LIN {X 0,Y 236.008,Z 310.681,A -85,B 0,C 180,E1 -19500.944,E2 -19500.944} C_VEL
LIN {X 0,Y 236.836,Z 313.931,A -85,B 0,C 180,E1 -19501.282,E2 -19501.282} C_VEL
LIN {X 0,Y 239.415,Z 324.062,A -85,B 0,C 180,E1 -19502.528,E2 -19502.528} C_VEL
LIN {X 0,Y 241.181,Z 333.604,A -85,B 0,C 180,E1 -19503.852,E2 -19503.852} C_VEL
LIN {X 0,Y 242.176,Z 341.797,A -85,B 0,C 180,E1 -19505.138,E2 -19505.138} C_VEL
LIN {X 0,Y 242.615,Z 349.643,A -85,B 0,C 180,E1 -19506.53,E2 -19506.53} C_VEL
LIN {X 0,Y 242.455,Z 357.246,A -85,B 0,C 180,E1 -19508.066,E2 -19508.066} C_VEL
LIN {X 0,Y 241.956,Z 362.587,A -85,B 0,C 180,E1 -19509.279,E2 -19509.279} C_VEL
LIN {X 0,Y 240.306,Z 368.641,A -85,B 0,C 180,E1 -19510.793,E2 -19510.793} C_VEL
LIN {X 0,Y 238.573,Z 374.082,A -85,B 0,C 180,E1 -19512.428,E2 -19512.428} C_VEL
LIN {X 0,Y 236.726,Z 379.604,A -85,B 0,C 180,E1 -19514.505,E2 -19514.505} C_VEL
LIN {X 0,Y 235.064,Z 384.766,A -85,B 0,C 180,E1 -19517.044,E2 -19517.044} C_VEL
LIN {X 0,Y 233.873,Z 388.583,A -85,B 0,C 180,E1 -19519.615,E2 -19519.615} C_VEL
LIN {X 0,Y 233.308,Z 390.355,A -85,B 0,C 180,E1 -19521.34,E2 -19521.34} C_VEL
LIN {X 0,Y 232.985,Z 391.647,A -85,B 0,C 180,E1 -19523.072,E2 -19523.072} C_VEL
LIN {X 0,Y 232.787,Z 392.537,A -85,B 0,C 180,E1 -19525.087,E2 -19525.087} C_VEL
LIN {X 0,Y 232.804,Z 392.826,A -85,B 0,C 180,E1 -19526.541,E2 -19526.541} C_VEL
LIN {X 0,Y 232.91,Z 392.585,A -85,B 0,C 180,E1 -19528.273,E2 -19528.273} C_VEL
LIN {X 0,Y 232.953,Z 391.86,A -85,B 0,C 180,E1 -19530.002,E2 -19530.002} C_VEL
LIN {X 0,Y 232.952,Z 390.653,A -85,B 0,C 180,E1 -19531.731,E2 -19531.731} C_VEL
LIN {X 0,Y 232.931,Z 388.936,A -85,B 0,C 180,E1 -19533.462,E2 -19533.462} C_VEL
LIN {X 0,Y 232.977,Z 385.143,A -85,B 0,C 180,E1 -19536.063,E2 -19536.063} C_VEL
LIN {X 0,Y 233.32,Z 379.947,A -85,B 0,C 180,E1 -19538.664,E2 -19538.664} C_VEL
LIN {X 0,Y 233.786,Z 374.337,A -85,B 0,C 180,E1 -19540.832,E2 -19540.832} C_VEL
LIN {X 0,Y 234.62,Z 367.267,A -85,B 0,C 180,E1 -19542.985,E2 -19542.985} C_VEL
LIN {X 0,Y 235.626,Z 359.155,A -85,B 0,C 180,E1 -19544.91,E2 -19544.91} C_VEL
LIN {X 0,Y 236.286,Z 352.615,A -85,B 0,C 180,E1 -19546.194,E2 -19546.194} C_VEL
LIN {X 0,Y 236.114,Z 344.809,A -85,B 0,C 180,E1 -19547.498,E2 -19547.498} C_VEL
LIN {X 0,Y 235.752,Z 335.886,A -85,B 0,C 180,E1 -19548.713,E2 -19548.713} C_VEL
LIN {X 0,Y 235.263,Z 327.406,A -85,B 0,C 180,E1 -19549.64,E2 -19549.64} C_VEL
LIN {X 0,Y 234.318,Z 317.752,A -85,B 0,C 180,E1 -19550.466,E2 -19550.466} C_VEL
LIN {X 0,Y 233.579,Z 311.732,A -85,B 0,C 180,E1 -19550.937,E2 -19550.937} C_VEL
LIN {X 0,Y 234.467,Z 305.559,A -85,B 0,C 180,E1 -19555.938,E2 -19555.938} C_VEL
LIN {X 0,Y 235.489,Z 299.992,A -85,B 0,C 180,E1 -19560.49,E2 -19560.49} C_VEL
LIN {X 0,Y 236.19,Z 296.337,A -85,B 0,C 180,E1 -19563.572,E2 -19563.572} C_VEL
LIN {X 0,Y 236.161,Z 294.216,A -85,B 0,C 180,E1 -19565.432,E2 -19565.432} C_VEL
LIN {X 0,Y 235.471,Z 290.233,A -85,B 0,C 180,E1 -19569.1,E2 -19569.1} C_VEL
LIN {X 0,Y 235.075,Z 288.016,A -85,B 0,C 180,E1 -19571.3,E2 -19571.3} C_VEL
LIN {X 0,Y 234.899,Z 288.035,A -85,B 0,C 180,E1 -19576.514,E2 -19576.514} C_VEL
LIN {X 0,Y 234.93,Z 288.031,A -85,B 0,C 180,E1 -19581.078,E2 -19581.078} C_VEL
LIN {X 0,Y 234.942,Z 288.032,A -85,B 0,C 180,E1 -19585.361,E2 -19585.361} C_VEL
LIN {X 0,Y 234.943,Z 288.029,A -85,B 0,C 180,E1 -19589.431,E2 -19589.431} C_VEL
LIN {X 0,Y 235.006,Z 288.023,A -85,B 0,C 180,E1 -19593.792,E2 -19593.792} C_VEL
LIN {X 0,Y 234.98,Z 288.022,A -85,B 0,C 180,E1 -19598.964,E2 -19598.964} C_VEL
LIN {X 0,Y 235.067,Z 288.018,A -85,B 0,C 180,E1 -19603.09,E2 -19603.09} C_VEL
LIN {X 0,Y 235.106,Z 288.003,A -85,B 0,C 180,E1 -19607.919,E2 -19607.919} C_VEL
LIN {X 0,Y 235.328,Z 287.982,A -85,B 0,C 180,E1 -19611.409,E2 -19611.409} C_VEL
LIN {X 0,Y 235.375,Z 287.978,A -85,B 0,C 180,E1 -19613.138,E2 -19613.138} C_VEL
LIN {X 0,Y 235.603,Z 287.945,A -85,B 0,C 180,E1 -19618.288,E2 -19618.288} C_VEL
LIN {X 0,Y 235.603,Z 287.946,A -85,B 0,C 180,E1 -19621.706,E2 -19621.706} C_VEL
LIN {X 0,Y 235.411,Z 287.971,A -85,B 0,C 180,E1 -19626.855,E2 -19626.855} C_VEL
LIN {X 0,Y 235.243,Z 287.989,A -85,B 0,C 180,E1 -19630.323,E2 -19630.323} C_VEL
LIN {X 0,Y 235.116,Z 288.009,A -85,B 0,C 180,E1 -19635.603,E2 -19635.603} C_VEL
LIN {X 0,Y 235.012,Z 288.02,A -85,B 0,C 180,E1 -19639.202,E2 -19639.202} C_VEL
LIN {X 0,Y 234.963,Z 288.023,A -85,B 0,C 180,E1 -19642.879,E2 -19642.879} C_VEL
LIN {X 0,Y 234.97,Z 288.027,A -85,B 0,C 180,E1 -19646.653,E2 -19646.653} C_VEL
LIN {X 0,Y 234.931,Z 288.031,A -85,B 0,C 180,E1 -19650.564,E2 -19650.564} C_VEL
LIN {X 0,Y 234.958,Z 288.027,A -85,B 0,C 180,E1 -19654.629,E2 -19654.629} C_VEL
LIN {X 0,Y 234.994,Z 288.025,A -85,B 0,C 180,E1 -19658.957,E2 -19658.957} C_VEL
LIN {X 0,Y 234.991,Z 288.027,A -85,B 0,C 180,E1 -19663.457,E2 -19663.457} C_VEL
LIN {X 0,Y 234.99,Z 288.024,A -85,B 0,C 180,E1 -19666.535,E2 -19666.535} C_VEL
LIN {X 0,Y 234.948,Z 288.032,A -85,B 0,C 180,E1 -19671.082,E2 -19671.082} C_VEL
LIN {X 0,Y 234.952,Z 288.03,A -85,B 0,C 180,E1 -19675.363,E2 -19675.363} C_VEL
LIN {X 0,Y 234.959,Z 288.029,A -85,B 0,C 180,E1 -19680.154,E2 -19680.154} C_VEL
LIN {X 0,Y 234.983,Z 288.025,A -85,B 0,C 180,E1 -19683.79,E2 -19683.79} C_VEL
LIN {X 0,Y 234.963,Z 288.028,A -85,B 0,C 180,E1 -19687.998,E2 -19687.998} C_VEL
LIN {X 0,Y 234.735,Z 288.058,A -85,B 0,C 180,E1 -19692.576,E2 -19692.576} C_VEL
LIN {X 0,Y 234.34,Z 288.106,A -85,B 0,C 180,E1 -19696.116,E2 -19696.116} C_VEL
LIN {X 0,Y 234.116,Z 288.347,A -85,B 0,C 180,E1 -19698.307,E2 -19698.307} C_VEL
LIN {X 0,Y 234.103,Z 291.422,A -85,B 0,C 180,E1 -19702.145,E2 -19702.145} C_VEL
LIN {X 0,Y 234.001,Z 292.577,A -85,B 0,C 180,E1 -19703.314,E2 -19703.314} C_VEL
LIN {X 0,Y 236.168,Z 303.411,A -85,B 0,C 180,E1 -19704.234,E2 -19704.234} C_VEL
LIN {X 0,Y 237.327,Z 311.672,A -85,B 0,C 180,E1 -19705.114,E2 -19705.114} C_VEL
LIN {X 0,Y 238.306,Z 321.335,A -85,B 0,C 180,E1 -19706.405,E2 -19706.405} C_VEL
LIN {X 0,Y 237.452,Z 329.525,A -85,B 0,C 180,E1 -19707.665,E2 -19707.665} C_VEL
LIN {X 0,Y 236.487,Z 337.321,A -85,B 0,C 180,E1 -19709.146,E2 -19709.146} C_VEL
LIN {X 0,Y 235.36,Z 346.28,A -85,B 0,C 180,E1 -19711.281,E2 -19711.281} C_VEL
LIN {X 0,Y 234.486,Z 353.183,A -85,B 0,C 180,E1 -19713.434,E2 -19713.434} C_VEL
LIN {X 0,Y 233.98,Z 357.734,A -85,B 0,C 180,E1 -19715.168,E2 -19715.168} C_VEL
LIN {X 0,Y 233.523,Z 361.536,A -85,B 0,C 180,E1 -19716.912,E2 -19716.912} C_VEL
LIN {X 0,Y 232.998,Z 365.862,A -85,B 0,C 180,E1 -19719.547,E2 -19719.547} C_VEL
LIN {X 0,Y 232.736,Z 368.898,A -85,B 0,C 180,E1 -19722.201,E2 -19722.201} C_VEL
LIN {X 0,Y 232.797,Z 370.803,A -85,B 0,C 180,E1 -19724.987,E2 -19724.987} C_VEL
LIN {X 0,Y 233.038,Z 371.385,A -85,B 0,C 180,E1 -19727.55,E2 -19727.55} C_VEL
LIN {X 0,Y 233.453,Z 371.103,A -85,B 0,C 180,E1 -19729.336,E2 -19729.336} C_VEL
LIN {X 0,Y 234.146,Z 370.082,A -85,B 0,C 180,E1 -19731.502,E2 -19731.502} C_VEL
LIN {X 0,Y 235.525,Z 367.076,A -85,B 0,C 180,E1 -19734.69,E2 -19734.69} C_VEL
LIN {X 0,Y 237.062,Z 363.279,A -85,B 0,C 180,E1 -19737.213,E2 -19737.213} C_VEL
LIN {X 0,Y 238.439,Z 359.51,A -85,B 0,C 180,E1 -19739.097,E2 -19739.097} C_VEL
LIN {X 0,Y 239.916,Z 355.184,A -85,B 0,C 180,E1 -19740.837,E2 -19740.837} C_VEL
LIN {X 0,Y 241.768,Z 349.341,A -85,B 0,C 180,E1 -19742.728,E2 -19742.728} C_VEL
LIN {X 0,Y 243.49,Z 343.538,A -85,B 0,C 180,E1 -19744.249,E2 -19744.249} C_VEL
LIN {X 0,Y 245.449,Z 336.245,A -85,B 0,C 180,E1 -19745.811,E2 -19745.811} C_VEL
LIN {X 0,Y 245.573,Z 333.35,A -85,B 0,C 180,E1 -19746.445,E2 -19746.445} C_VEL
LIN {X 0,Y 244.381,Z 324.378,A -85,B 0,C 180,E1 -19748.274,E2 -19748.274} C_VEL
LIN {X 0,Y 242.509,Z 315.823,A -85,B 0,C 180,E1 -19749.832,E2 -19749.832} C_VEL
LIN {X 0,Y 240.136,Z 307.625,A -85,B 0,C 180,E1 -19751.189,E2 -19751.189} C_VEL
LIN {X 0,Y 236.731,Z 298.443,A -85,B 0,C 180,E1 -19752.592,E2 -19752.592} C_VEL
LIN {X 0,Y 235.009,Z 293.938,A -85,B 0,C 180,E1 -19753.227,E2 -19753.227} C_VEL
LIN {X 0,Y 234.961,Z 293.585,A -85,B 0,C 180,E1 -19753.299,E2 -19753.299} C_VEL
LIN {X 0,Y 235.134,Z 291.455,A -85,B 0,C 180,E1 -19756.576,E2 -19756.576} C_VEL
LIN {X 0,Y 235.094,Z 290.036,A -85,B 0,C 180,E1 -19758.882,E2 -19758.882} C_VEL
LIN {X 0,Y 235.006,Z 288.731,A -85,B 0,C 180,E1 -19761.101,E2 -19761.101} C_VEL
LIN {X 0,Y 234.937,Z 288.037,A -85,B 0,C 180,E1 -19763.866,E2 -19763.866} C_VEL
LIN {X 0,Y 234.943,Z 288.032,A -85,B 0,C 180,E1 -19767.427,E2 -19767.427} C_VEL
LIN {X 0,Y 234.919,Z 288.033,A -85,B 0,C 180,E1 -19771.406,E2 -19771.406} C_VEL
LIN {X 0,Y 234.963,Z 288.03,A -85,B 0,C 180,E1 -19775.248,E2 -19775.248} C_VEL
LIN {X 0,Y 234.983,Z 288.023,A -85,B 0,C 180,E1 -19778.971,E2 -19778.971} C_VEL
LIN {X 0,Y 235.082,Z 288.011,A -85,B 0,C 180,E1 -19783.062,E2 -19783.062} C_VEL
LIN {X 0,Y 235.13,Z 288.01,A -85,B 0,C 180,E1 -19787.926,E2 -19787.926} C_VEL
LIN {X 0,Y 235.309,Z 287.988,A -85,B 0,C 180,E1 -19791.415,E2 -19791.415} C_VEL
LIN {X 0,Y 235.347,Z 287.975,A -85,B 0,C 180,E1 -19793.143,E2 -19793.143} C_VEL
LIN {X 0,Y 235.586,Z 287.945,A -85,B 0,C 180,E1 -19798.294,E2 -19798.294} C_VEL
LIN {X 0,Y 235.586,Z 287.945,A -85,B 0,C 180,E1 -19801.713,E2 -19801.713} C_VEL
LIN {X 0,Y 235.397,Z 287.97,A -85,B 0,C 180,E1 -19806.862,E2 -19806.862} C_VEL
LIN {X 0,Y 235.246,Z 287.996,A -85,B 0,C 180,E1 -19810.329,E2 -19810.329} C_VEL
LIN {X 0,Y 235.107,Z 288.012,A -85,B 0,C 180,E1 -19815.61,E2 -19815.61} C_VEL
LIN {X 0,Y 235.002,Z 288.025,A -85,B 0,C 180,E1 -19819.209,E2 -19819.209} C_VEL
LIN {X 0,Y 234.941,Z 288.036,A -85,B 0,C 180,E1 -19822.888,E2 -19822.888} C_VEL
LIN {X 0,Y 234.94,Z 288.037,A -85,B 0,C 180,E1 -19826.664,E2 -19826.664} C_VEL
LIN {X 0,Y 234.895,Z 288.046,A -85,B 0,C 180,E1 -19830.576,E2 -19830.576} C_VEL
LIN {X 0,Y 234.957,Z 288.038,A -85,B 0,C 180,E1 -19834.636,E2 -19834.636} C_VEL
LIN {X 0,Y 234.993,Z 288.035,A -85,B 0,C 180,E1 -19836.153,E2 -19836.153} C_VEL
LIN {X 0,Y 235.324,Z 290.078,A -85,B 0,C 180,E1 -19839.063,E2 -19839.063} C_VEL
LIN {X 0,Y 235.81,Z 293.316,A -85,B 0,C 180,E1 -19843.277,E2 -19843.277} C_VEL
LIN {X 0,Y 236.483,Z 297.318,A -85,B 0,C 180,E1 -19847.988,E2 -19847.988} C_VEL
LIN {X 0,Y 237.095,Z 300.545,A -85,B 0,C 180,E1 -19851.505,E2 -19851.505} C_VEL
LIN {X 0,Y 237.449,Z 303.212,A -85,B 0,C 180,E1 -19854.2,E2 -19854.2} C_VEL
LIN {X 0,Y 236.801,Z 304.253,A -85,B 0,C 180,E1 -19855.103,E2 -19855.103} C_VEL
LIN {X 0,Y 233.819,Z 306.165,A -85,B 0,C 180,E1 -19856.484,E2 -19856.484} C_VEL
LIN {X 0,Y 230.582,Z 308.119,A -85,B 0,C 180,E1 -19857.893,E2 -19857.893} C_VEL
LIN {X 0,Y 229.602,Z 309.245,A -85,B 0,C 180,E1 -19858.83,E2 -19858.83} C_VEL
LIN {X 0,Y 229.293,Z 310.304,A -85,B 0,C 180,E1 -19859.784,E2 -19859.784} C_VEL
LIN {X 0,Y 230.185,Z 313.716,A -85,B 0,C 180,E1 -19860.165,E2 -19860.165} C_VEL
LIN {X 0,Y 232.856,Z 324.19,A -85,B 0,C 180,E1 -19861.531,E2 -19861.531} C_VEL
LIN {X 0,Y 234.553,Z 333.427,A -85,B 0,C 180,E1 -19862.882,E2 -19862.882} C_VEL
LIN {X 0,Y 235.447,Z 340.923,A -85,B 0,C 180,E1 -19864.102,E2 -19864.102} C_VEL
LIN {X 0,Y 236.011,Z 349.022,A -85,B 0,C 180,E1 -19865.598,E2 -19865.598} C_VEL
LIN {X 0,Y 235.901,Z 356.764,A -85,B 0,C 180,E1 -19867.216,E2 -19867.216} C_VEL
LIN {X 0,Y 235.274,Z 362.992,A -85,B 0,C 180,E1 -19868.693,E2 -19868.693} C_VEL
LIN {X 0,Y 233.628,Z 368.826,A -85,B 0,C 180,E1 -19870.222,E2 -19870.222} C_VEL
LIN {X 0,Y 231.835,Z 374.177,A -85,B 0,C 180,E1 -19871.9,E2 -19871.9} C_VEL
LIN {X 0,Y 229.886,Z 379.621,A -85,B 0,C 180,E1 -19874.032,E2 -19874.032} C_VEL
LIN {X 0,Y 228.141,Z 384.711,A -85,B 0,C 180,E1 -19876.644,E2 -19876.644} C_VEL
LIN {X 0,Y 226.878,Z 388.454,A -85,B 0,C 180,E1 -19879.291,E2 -19879.291} C_VEL
LIN {X 0,Y 226.285,Z 390.169,A -85,B 0,C 180,E1 -19881.069,E2 -19881.069} C_VEL
LIN {X 0,Y 225.927,Z 391.401,A -85,B 0,C 180,E1 -19882.855,E2 -19882.855} C_VEL
LIN {X 0,Y 225.706,Z 392.282,A -85,B 0,C 180,E1 -19885.167,E2 -19885.167} C_VEL
LIN {X 0,Y 225.709,Z 392.49,A -85,B 0,C 180,E1 -19886.432,E2 -19886.432} C_VEL
LIN {X 0,Y 225.838,Z 392.227,A -85,B 0,C 180,E1 -19888.219,E2 -19888.219} C_VEL
LIN {X 0,Y 225.882,Z 391.447,A -85,B 0,C 180,E1 -19890.002,E2 -19890.002} C_VEL
LIN {X 0,Y 225.882,Z 390.182,A -85,B 0,C 180,E1 -19891.785,E2 -19891.785} C_VEL
LIN {X 0,Y 225.789,Z 387.389,A -85,B 0,C 180,E1 -19894.352,E2 -19894.352} C_VEL
LIN {X 0,Y 225.918,Z 384.546,A -85,B 0,C 180,E1 -19896.253,E2 -19896.253} C_VEL
LIN {X 0,Y 226.11,Z 381.21,A -85,B 0,C 180,E1 -19898.043,E2 -19898.043} C_VEL
LIN {X 0,Y 226.472,Z 377.155,A -85,B 0,C 180,E1 -19899.83,E2 -19899.83} C_VEL
LIN {X 0,Y 227.131,Z 370.824,A -85,B 0,C 180,E1 -19902.058,E2 -19902.058} C_VEL
LIN {X 0,Y 227.879,Z 364.62,A -85,B 0,C 180,E1 -19903.831,E2 -19903.831} C_VEL
LIN {X 0,Y 228.776,Z 358.107,A -85,B 0,C 180,E1 -19905.367,E2 -19905.367} C_VEL
LIN {X 0,Y 229.258,Z 352.645,A -85,B 0,C 180,E1 -19906.475,E2 -19906.475} C_VEL
LIN {X 0,Y 229.055,Z 343.894,A -85,B 0,C 180,E1 -19907.974,E2 -19907.974} C_VEL
LIN {X 0,Y 228.8,Z 336.258,A -85,B 0,C 180,E1 -19909.05,E2 -19909.05} C_VEL
LIN {X 0,Y 228.248,Z 326.901,A -85,B 0,C 180,E1 -19910.111,E2 -19910.111} C_VEL
LIN {X 0,Y 227.293,Z 317.696,A -85,B 0,C 180,E1 -19910.93,E2 -19910.93} C_VEL
LIN {X 0,Y 226.538,Z 311.466,A -85,B 0,C 180,E1 -19911.381,E2 -19911.381} C_VEL
LIN {X 0,Y 227.302,Z 306.394,A -85,B 0,C 180,E1 -19915.652,E2 -19915.652} C_VEL
LIN {X 0,Y 228.394,Z 300.678,A -85,B 0,C 180,E1 -19920.499,E2 -19920.499} C_VEL
LIN {X 0,Y 229.108,Z 297.178,A -85,B 0,C 180,E1 -19923.518,E2 -19923.518} C_VEL
LIN {X 0,Y 229.089,Z 294.828,A -85,B 0,C 180,E1 -19925.656,E2 -19925.656} C_VEL
LIN {X 0,Y 228.228,Z 289.995,A -85,B 0,C 180,E1 -19930.293,E2 -19930.293} C_VEL
LIN {X 0,Y 227.996,Z 288.898,A -85,B 0,C 180,E1 -19931.512,E2 -19931.512} C_VEL
LIN {X 0,Y 227.846,Z 288.914,A -85,B 0,C 180,E1 -19935.192,E2 -19935.192} C_VEL
LIN {X 0,Y 227.838,Z 288.918,A -85,B 0,C 180,E1 -19939.623,E2 -19939.623} C_VEL
LIN {X 0,Y 227.893,Z 288.909,A -85,B 0,C 180,E1 -19944.127,E2 -19944.127} C_VEL
LIN {X 0,Y 227.882,Z 288.906,A -85,B 0,C 180,E1 -19948.377,E2 -19948.377} C_VEL
LIN {X 0,Y 227.898,Z 288.907,A -85,B 0,C 180,E1 -19952.444,E2 -19952.444} C_VEL
LIN {X 0,Y 227.917,Z 288.902,A -85,B 0,C 180,E1 -19956.365,E2 -19956.365} C_VEL
LIN {X 0,Y 227.925,Z 288.902,A -85,B 0,C 180,E1 -19960.17,E2 -19960.17} C_VEL
LIN {X 0,Y 228.031,Z 288.891,A -85,B 0,C 180,E1 -19963.893,E2 -19963.893} C_VEL
LIN {X 0,Y 228.064,Z 288.881,A -85,B 0,C 180,E1 -19967.54,E2 -19967.54} C_VEL
LIN {X 0,Y 228.26,Z 288.864,A -85,B 0,C 180,E1 -19971.141,E2 -19971.141} C_VEL
LIN {X 0,Y 228.325,Z 288.858,A -85,B 0,C 180,E1 -19972.925,E2 -19972.925} C_VEL
LIN {X 0,Y 228.561,Z 288.822,A -85,B 0,C 180,E1 -19978.235,E2 -19978.235} C_VEL
LIN {X 0,Y 228.562,Z 288.823,A -85,B 0,C 180,E1 -19981.759,E2 -19981.759} C_VEL
LIN {X 0,Y 228.361,Z 288.849,A -85,B 0,C 180,E1 -19987.068,E2 -19987.068} C_VEL
LIN {X 0,Y 228.169,Z 288.87,A -85,B 0,C 180,E1 -19990.647,E2 -19990.647} C_VEL
LIN {X 0,Y 228.067,Z 288.889,A -85,B 0,C 180,E1 -19994.268,E2 -19994.268} C_VEL
LIN {X 0,Y 228.007,Z 288.897,A -85,B 0,C 180,E1 -19997.949,E2 -19997.949} C_VEL
LIN {X 0,Y 227.932,Z 288.9,A -85,B 0,C 180,E1 -20002.325,E2 -20002.325} C_VEL
LIN {X 0,Y 227.943,Z 288.902,A -85,B 0,C 180,E1 -20006.598,E2 -20006.598} C_VEL
LIN {X 0,Y 227.907,Z 288.906,A -85,B 0,C 180,E1 -20010.291,E2 -20010.291} C_VEL
LIN {X 0,Y 227.888,Z 288.911,A -85,B 0,C 180,E1 -20013.714,E2 -20013.714} C_VEL
LIN {X 0,Y 227.888,Z 288.91,A -85,B 0,C 180,E1 -20018.077,E2 -20018.077} C_VEL
LIN {X 0,Y 227.931,Z 288.904,A -85,B 0,C 180,E1 -20022.709,E2 -20022.709} C_VEL
LIN {X 0,Y 227.923,Z 288.908,A -85,B 0,C 180,E1 -20027.281,E2 -20027.281} C_VEL
LIN {X 0,Y 227.864,Z 288.912,A -85,B 0,C 180,E1 -20031.91,E2 -20031.91} C_VEL
LIN {X 0,Y 227.881,Z 288.911,A -85,B 0,C 180,E1 -20036.369,E2 -20036.369} C_VEL
LIN {X 0,Y 227.909,Z 288.908,A -85,B 0,C 180,E1 -20040.434,E2 -20040.434} C_VEL
LIN {X 0,Y 227.917,Z 288.908,A -85,B 0,C 180,E1 -20044.422,E2 -20044.422} C_VEL
LIN {X 0,Y 227.921,Z 288.907,A -85,B 0,C 180,E1 -20048.281,E2 -20048.281} C_VEL
LIN {X 0,Y 227.668,Z 288.937,A -85,B 0,C 180,E1 -20053.113,E2 -20053.113} C_VEL
LIN {X 0,Y 227.073,Z 289.046,A -85,B 0,C 180,E1 -20058.166,E2 -20058.166} C_VEL
LIN {X 0,Y 226.974,Z 292.656,A -85,B 0,C 180,E1 -20062.791,E2 -20062.791} C_VEL
LIN {X 0,Y 229.271,Z 304.335,A -85,B 0,C 180,E1 -20063.839,E2 -20063.839} C_VEL
LIN {X 0,Y 230.419,Z 312.457,A -85,B 0,C 180,E1 -20064.748,E2 -20064.748} C_VEL
LIN {X 0,Y 231.205,Z 320.636,A -85,B 0,C 180,E1 -20065.858,E2 -20065.858} C_VEL
LIN {X 0,Y 231.077,Z 325.043,A -85,B 0,C 180,E1 -20066.51,E2 -20066.51} C_VEL
LIN {X 0,Y 229.823,Z 334.841,A -85,B 0,C 180,E1 -20068.245,E2 -20068.245} C_VEL
LIN {X 0,Y 228.881,Z 342.581,A -85,B 0,C 180,E1 -20069.998,E2 -20069.998} C_VEL
LIN {X 0,Y 228.019,Z 348.96,A -85,B 0,C 180,E1 -20071.764,E2 -20071.764} C_VEL
LIN {X 0,Y 227.352,Z 354.255,A -85,B 0,C 180,E1 -20073.542,E2 -20073.542} C_VEL
LIN {X 0,Y 226.845,Z 358.671,A -85,B 0,C 180,E1 -20075.331,E2 -20075.331} C_VEL
LIN {X 0,Y 226.377,Z 362.354,A -85,B 0,C 180,E1 -20077.131,E2 -20077.131} C_VEL
LIN {X 0,Y 226.018,Z 365.378,A -85,B 0,C 180,E1 -20078.942,E2 -20078.942} C_VEL
LIN {X 0,Y 225.749,Z 367.747,A -85,B 0,C 180,E1 -20080.763,E2 -20080.763} C_VEL
LIN {X 0,Y 225.632,Z 369.493,A -85,B 0,C 180,E1 -20082.591,E2 -20082.591} C_VEL
LIN {X 0,Y 225.729,Z 371.137,A -85,B 0,C 180,E1 -20085.182,E2 -20085.182} C_VEL
LIN {X 0,Y 226.064,Z 371.688,A -85,B 0,C 180,E1 -20088.11,E2 -20088.11} C_VEL
LIN {X 0,Y 226.529,Z 371.38,A -85,B 0,C 180,E1 -20089.952,E2 -20089.952} C_VEL
LIN {X 0,Y 227.194,Z 370.422,A -85,B 0,C 180,E1 -20091.884,E2 -20091.884} C_VEL
LIN {X 0,Y 227.911,Z 369.033,A -85,B 0,C 180,E1 -20093.63,E2 -20093.63} C_VEL
LIN {X 0,Y 229.383,Z 365.869,A -85,B 0,C 180,E1 -20096.373,E2 -20096.373} C_VEL
LIN {X 0,Y 231.271,Z 361.194,A -85,B 0,C 180,E1 -20099.089,E2 -20099.089} C_VEL
LIN {X 0,Y 233.181,Z 355.971,A -85,B 0,C 180,E1 -20101.323,E2 -20101.323} C_VEL
LIN {X 0,Y 234.93,Z 350.723,A -85,B 0,C 180,E1 -20103.117,E2 -20103.117} C_VEL
LIN {X 0,Y 236.883,Z 344.532,A -85,B 0,C 180,E1 -20104.825,E2 -20104.825} C_VEL
LIN {X 0,Y 238.87,Z 337.589,A -85,B 0,C 180,E1 -20106.379,E2 -20106.379} C_VEL
LIN {X 0,Y 239.035,Z 335.431,A -85,B 0,C 180,E1 -20106.869,E2 -20106.869} C_VEL
LIN {X 0,Y 237.849,Z 325.521,A -85,B 0,C 180,E1 -20109.034,E2 -20109.034} C_VEL
LIN {X 0,Y 236.096,Z 317.291,A -85,B 0,C 180,E1 -20110.625,E2 -20110.625} C_VEL
LIN {X 0,Y 233.545,Z 308.548,A -85,B 0,C 180,E1 -20112.165,E2 -20112.165} C_VEL
LIN {X 0,Y 230.284,Z 299.911,A -85,B 0,C 180,E1 -20113.588,E2 -20113.588} C_VEL
LIN {X 0,Y 228.115,Z 294.568,A -85,B 0,C 180,E1 -20114.413,E2 -20114.413} C_VEL
LIN {X 0,Y 228.023,Z 293.993,A -85,B 0,C 180,E1 -20114.508,E2 -20114.508} C_VEL
LIN {X 0,Y 228.108,Z 292.023,A -85,B 0,C 180,E1 -20117.68,E2 -20117.68} C_VEL
LIN {X 0,Y 227.928,Z 289.589,A -85,B 0,C 180,E1 -20121.931,E2 -20121.931} C_VEL
LIN {X 0,Y 227.886,Z 288.915,A -85,B 0,C 180,E1 -20123.302,E2 -20123.302} C_VEL
LIN {X 0,Y 227.873,Z 288.914,A -85,B 0,C 180,E1 -20126.375,E2 -20126.375} C_VEL
LIN {X 0,Y 227.888,Z 288.912,A -85,B 0,C 180,E1 -20130.438,E2 -20130.438} C_VEL
LIN {X 0,Y 227.909,Z 288.909,A -85,B 0,C 180,E1 -20134.428,E2 -20134.428} C_VEL
LIN {X 0,Y 227.933,Z 288.904,A -85,B 0,C 180,E1 -20138.288,E2 -20138.288} C_VEL
LIN {X 0,Y 228.021,Z 288.889,A -85,B 0,C 180,E1 -20142.828,E2 -20142.828} C_VEL
LIN {X 0,Y 228.079,Z 288.888,A -85,B 0,C 180,E1 -20147.547,E2 -20147.547} C_VEL
LIN {X 0,Y 228.247,Z 288.865,A -85,B 0,C 180,E1 -20151.147,E2 -20151.147} C_VEL
LIN {X 0,Y 228.299,Z 288.854,A -85,B 0,C 180,E1 -20152.93,E2 -20152.93} C_VEL
LIN {X 0,Y 228.544,Z 288.822,A -85,B 0,C 180,E1 -20158.241,E2 -20158.241} C_VEL
LIN {X 0,Y 228.545,Z 288.822,A -85,B 0,C 180,E1 -20161.765,E2 -20161.765} C_VEL
LIN {X 0,Y 228.349,Z 288.849,A -85,B 0,C 180,E1 -20167.075,E2 -20167.075} C_VEL
LIN {X 0,Y 228.164,Z 288.877,A -85,B 0,C 180,E1 -20170.653,E2 -20170.653} C_VEL
LIN {X 0,Y 228.051,Z 288.892,A -85,B 0,C 180,E1 -20176.106,E2 -20176.106} C_VEL
LIN {X 0,Y 227.931,Z 288.906,A -85,B 0,C 180,E1 -20179.829,E2 -20179.829} C_VEL
LIN {X 0,Y 227.89,Z 288.912,A -85,B 0,C 180,E1 -20183.638,E2 -20183.638} C_VEL
LIN {X 0,Y 227.85,Z 288.922,A -85,B 0,C 180,E1 -20187.563,E2 -20187.563} C_VEL
LIN {X 0,Y 227.854,Z 288.922,A -85,B 0,C 180,E1 -20191.628,E2 -20191.628} C_VEL
LIN {X 0,Y 227.979,Z 289.073,A -85,B 0,C 180,E1 -20195.314,E2 -20195.314} C_VEL
LIN {X 0,Y 228.451,Z 292.089,A -85,B 0,C 180,E1 -20199.732,E2 -20199.732} C_VEL
LIN {X 0,Y 228.754,Z 294.17,A -85,B 0,C 180,E1 -20202.528,E2 -20202.528} C_VEL
LIN {X 0,Y 229.419,Z 298.061,A -85,B 0,C 180,E1 -20207.329,E2 -20207.329} C_VEL
LIN {X 0,Y 230.072,Z 301.512,A -85,B 0,C 180,E1 -20211.232,E2 -20211.232} C_VEL
LIN {X 0,Y 230.496,Z 304.747,A -85,B 0,C 180,E1 -20214.6,E2 -20214.6} C_VEL
LIN {X 0,Y 229.965,Z 307.974,A -85,B 0,C 180,E1 -20217.671,E2 -20217.671} C_VEL
LIN {X 0,Y 229.602,Z 309.245,A -85,B 0,C 180,E1 -20218.83,E2 -20218.83} C_VEL
LIN {X 0,Y 229.759,Z 310.473,A -85,B 0,C 180,E1 -20219.478,E2 -20219.478} C_VEL
LIN {X 0,Y 230.705,Z 313.064,A -85,B 0,C 180,E1 -20220.17,E2 -20220.17} C_VEL
LIN {X 0,Y 232.123,Z 317.253,A -85,B 0,C 180,E1 -20220.774,E2 -20220.774} C_VEL
LIN {X 0,Y 232.473,Z 321.036,A -85,B 0,C 180,E1 -20221.139,E2 -20221.139} C_VEL
LIN {X 0,Y 231.641,Z 325.307,A -85,B 0,C 180,E1 -20221.418,E2 -20221.418} C_VEL
LIN {X 0,Y 228.832,Z 333.716,A -85,B 0,C 180,E1 -20222.039,E2 -20222.039} C_VEL
LIN {X 0,Y 228.581,Z 337.299,A -85,B 0,C 180,E1 -20222.511,E2 -20222.511} C_VEL
LIN {X 0,Y 229.384,Z 347.335,A -85,B 0,C 180,E1 -20224.378,E2 -20224.378} C_VEL
LIN {X 0,Y 229.364,Z 355.19,A -85,B 0,C 180,E1 -20226.049,E2 -20226.049} C_VEL
LIN {X 0,Y 228.754,Z 362.606,A -85,B 0,C 180,E1 -20227.864,E2 -20227.864} C_VEL
LIN {X 0,Y 227.495,Z 367.593,A -85,B 0,C 180,E1 -20229.193,E2 -20229.193} C_VEL
LIN {X 0,Y 225.113,Z 374.273,A -85,B 0,C 180,E1 -20231.34,E2 -20231.34} C_VEL
LIN {X 0,Y 223.058,Z 379.638,A -85,B 0,C 180,E1 -20233.529,E2 -20233.529} C_VEL
LIN {X 0,Y 221.774,Z 383.127,A -85,B 0,C 180,E1 -20235.317,E2 -20235.317} C_VEL
LIN {X 0,Y 220.256,Z 387.171,A -85,B 0,C 180,E1 -20238.032,E2 -20238.032} C_VEL
LIN {X 0,Y 219.253,Z 389.985,A -85,B 0,C 180,E1 -20240.78,E2 -20240.78} C_VEL
LIN {X 0,Y 218.864,Z 391.157,A -85,B 0,C 180,E1 -20242.623,E2 -20242.623} C_VEL
LIN {X 0,Y 218.61,Z 392.038,A -85,B 0,C 180,E1 -20245.305,E2 -20245.305} C_VEL
LIN {X 0,Y 218.743,Z 391.866,A -85,B 0,C 180,E1 -20248.161,E2 -20248.161} C_VEL
LIN {X 0,Y 218.814,Z 391.03,A -85,B 0,C 180,E1 -20250.002,E2 -20250.002} C_VEL
LIN {X 0,Y 218.814,Z 389.706,A -85,B 0,C 180,E1 -20251.843,E2 -20251.843} C_VEL
LIN {X 0,Y 218.743,Z 387.861,A -85,B 0,C 180,E1 -20253.687,E2 -20253.687} C_VEL
LIN {X 0,Y 218.747,Z 385.462,A -85,B 0,C 180,E1 -20255.533,E2 -20255.533} C_VEL
LIN {X 0,Y 218.944,Z 382.399,A -85,B 0,C 180,E1 -20257.379,E2 -20257.379} C_VEL
LIN {X 0,Y 219.434,Z 376.391,A -85,B 0,C 180,E1 -20260.148,E2 -20260.148} C_VEL
LIN {X 0,Y 219.994,Z 371.404,A -85,B 0,C 180,E1 -20261.987,E2 -20261.987} C_VEL
LIN {X 0,Y 220.719,Z 365.379,A -85,B 0,C 180,E1 -20263.819,E2 -20263.819} C_VEL
LIN {X 0,Y 221.765,Z 358.054,A -85,B 0,C 180,E1 -20265.629,E2 -20265.629} C_VEL
LIN {X 0,Y 222.237,Z 352.764,A -85,B 0,C 180,E1 -20266.752,E2 -20266.752} C_VEL
LIN {X 0,Y 222.049,Z 343.105,A -85,B 0,C 180,E1 -20268.454,E2 -20268.454} C_VEL
LIN {X 0,Y 221.749,Z 334.464,A -85,B 0,C 180,E1 -20269.681,E2 -20269.681} C_VEL
LIN {X 0,Y 221.197,Z 326.273,A -85,B 0,C 180,E1 -20270.626,E2 -20270.626} C_VEL
LIN {X 0,Y 220.314,Z 317.035,A -85,B 0,C 180,E1 -20271.465,E2 -20271.465} C_VEL
LIN {X 0,Y 219.524,Z 311.153,A -85,B 0,C 180,E1 -20271.917,E2 -20271.917} C_VEL
LIN {X 0,Y 220.441,Z 305.581,A -85,B 0,C 180,E1 -20276.783,E2 -20276.783} C_VEL
LIN {X 0,Y 221.456,Z 300.736,A -85,B 0,C 180,E1 -20281.03,E2 -20281.03} C_VEL
LIN {X 0,Y 222.059,Z 297.866,A -85,B 0,C 180,E1 -20283.591,E2 -20283.591} C_VEL
LIN {X 0,Y 222.02,Z 295.475,A -85,B 0,C 180,E1 -20285.849,E2 -20285.849} C_VEL
LIN {X 0,Y 221.217,Z 290.975,A -85,B 0,C 180,E1 -20290.314,E2 -20290.314} C_VEL
LIN {X 0,Y 220.935,Z 289.778,A -85,B 0,C 180,E1 -20291.701,E2 -20291.701} C_VEL
LIN {X 0,Y 220.786,Z 289.794,A -85,B 0,C 180,E1 -20295.546,E2 -20295.546} C_VEL
LIN {X 0,Y 220.819,Z 289.789,A -85,B 0,C 180,E1 -20300.462,E2 -20300.462} C_VEL
LIN {X 0,Y 220.813,Z 289.791,A -85,B 0,C 180,E1 -20305.044,E2 -20305.044} C_VEL
LIN {X 0,Y 220.881,Z 289.78,A -85,B 0,C 180,E1 -20309.394,E2 -20309.394} C_VEL
LIN {X 0,Y 220.907,Z 289.781,A -85,B 0,C 180,E1 -20313.548,E2 -20313.548} C_VEL
LIN {X 0,Y 220.875,Z 289.778,A -85,B 0,C 180,E1 -20317.55,E2 -20317.55} C_VEL
LIN {X 0,Y 220.939,Z 289.775,A -85,B 0,C 180,E1 -20322.616,E2 -20322.616} C_VEL
LIN {X 0,Y 221.002,Z 289.762,A -85,B 0,C 180,E1 -20327.135,E2 -20327.135} C_VEL
LIN {X 0,Y 221.197,Z 289.743,A -85,B 0,C 180,E1 -20330.856,E2 -20330.856} C_VEL
LIN {X 0,Y 221.26,Z 289.737,A -85,B 0,C 180,E1 -20332.697,E2 -20332.697} C_VEL
LIN {X 0,Y 221.519,Z 289.699,A -85,B 0,C 180,E1 -20338.179,E2 -20338.179} C_VEL
LIN {X 0,Y 221.52,Z 289.7,A -85,B 0,C 180,E1 -20341.815,E2 -20341.815} C_VEL
LIN {X 0,Y 221.296,Z 289.728,A -85,B 0,C 180,E1 -20347.295,E2 -20347.295} C_VEL
LIN {X 0,Y 221.117,Z 289.747,A -85,B 0,C 180,E1 -20350.99,E2 -20350.99} C_VEL
LIN {X 0,Y 221.02,Z 289.765,A -85,B 0,C 180,E1 -20356.626,E2 -20356.626} C_VEL
LIN {X 0,Y 220.895,Z 289.775,A -85,B 0,C 180,E1 -20360.482,E2 -20360.482} C_VEL
LIN {X 0,Y 220.869,Z 289.783,A -85,B 0,C 180,E1 -20364.431,E2 -20364.431} C_VEL
LIN {X 0,Y 220.836,Z 289.787,A -85,B 0,C 180,E1 -20368.509,E2 -20368.509} C_VEL
LIN {X 0,Y 220.823,Z 289.789,A -85,B 0,C 180,E1 -20372.75,E2 -20372.75} C_VEL
LIN {X 0,Y 220.865,Z 289.786,A -85,B 0,C 180,E1 -20377.294,E2 -20377.294} C_VEL
LIN {X 0,Y 220.874,Z 289.783,A -85,B 0,C 180,E1 -20381.923,E2 -20381.923} C_VEL
LIN {X 0,Y 220.869,Z 289.785,A -85,B 0,C 180,E1 -20385.567,E2 -20385.567} C_VEL
LIN {X 0,Y 220.852,Z 289.785,A -85,B 0,C 180,E1 -20389.788,E2 -20389.788} C_VEL
LIN {X 0,Y 220.827,Z 289.791,A -85,B 0,C 180,E1 -20392.791,E2 -20392.791} C_VEL
LIN {X 0,Y 220.815,Z 289.791,A -85,B 0,C 180,E1 -20397.241,E2 -20397.241} C_VEL
LIN {X 0,Y 220.826,Z 289.788,A -85,B 0,C 180,E1 -20401.483,E2 -20401.483} C_VEL
LIN {X 0,Y 220.855,Z 289.785,A -85,B 0,C 180,E1 -20405.561,E2 -20405.561} C_VEL
LIN {X 0,Y 220.804,Z 289.792,A -85,B 0,C 180,E1 -20409.503,E2 -20409.503} C_VEL
LIN {X 0,Y 220.602,Z 289.817,A -85,B 0,C 180,E1 -20413.336,E2 -20413.336} C_VEL
LIN {X 0,Y 220.038,Z 289.928,A -85,B 0,C 180,E1 -20418.249,E2 -20418.249} C_VEL
LIN {X 0,Y 219.974,Z 292.962,A -85,B 0,C 180,E1 -20422.241,E2 -20422.241} C_VEL
LIN {X 0,Y 222.394,Z 305.255,A -85,B 0,C 180,E1 -20423.42,E2 -20423.42} C_VEL
LIN {X 0,Y 223.702,Z 314.98,A -85,B 0,C 180,E1 -20424.59,E2 -20424.59} C_VEL
LIN {X 0,Y 224.379,Z 322.752,A -85,B 0,C 180,E1 -20425.732,E2 -20425.732} C_VEL
LIN {X 0,Y 223.483,Z 330.802,A -85,B 0,C 180,E1 -20427.068,E2 -20427.068} C_VEL
LIN {X 0,Y 222.378,Z 339.511,A -85,B 0,C 180,E1 -20428.866,E2 -20428.866} C_VEL
LIN {X 0,Y 221.28,Z 347.314,A -85,B 0,C 180,E1 -20430.908,E2 -20430.908} C_VEL
LIN {X 0,Y 220.354,Z 354.137,A -85,B 0,C 180,E1 -20433.197,E2 -20433.197} C_VEL
LIN {X 0,Y 219.907,Z 357.654,A -85,B 0,C 180,E1 -20434.58,E2 -20434.58} C_VEL
LIN {X 0,Y 219.235,Z 363.165,A -85,B 0,C 180,E1 -20437.365,E2 -20437.365} C_VEL
LIN {X 0,Y 218.728,Z 367.265,A -85,B 0,C 180,E1 -20440.176,E2 -20440.176} C_VEL
LIN {X 0,Y 218.546,Z 370.087,A -85,B 0,C 180,E1 -20443.007,E2 -20443.007} C_VEL
LIN {X 0,Y 218.639,Z 371.46,A -85,B 0,C 180,E1 -20445.366,E2 -20445.366} C_VEL
LIN {X 0,Y 219.087,Z 371.975,A -85,B 0,C 180,E1 -20448.708,E2 -20448.708} C_VEL
LIN {X 0,Y 219.637,Z 371.609,A -85,B 0,C 180,E1 -20450.606,E2 -20450.606} C_VEL
LIN {X 0,Y 220.34,Z 370.654,A -85,B 0,C 180,E1 -20452.502,E2 -20452.502} C_VEL
LIN {X 0,Y 221.635,Z 368.183,A -85,B 0,C 180,E1 -20455.343,E2 -20455.343} C_VEL
LIN {X 0,Y 222.768,Z 365.816,A -85,B 0,C 180,E1 -20457.22,E2 -20457.22} C_VEL
LIN {X 0,Y 224.823,Z 360.913,A -85,B 0,C 180,E1 -20460.008,E2 -20460.008} C_VEL
LIN {X 0,Y 226.439,Z 356.757,A -85,B 0,C 180,E1 -20461.842,E2 -20461.842} C_VEL
LIN {X 0,Y 228.477,Z 351.038,A -85,B 0,C 180,E1 -20463.855,E2 -20463.855} C_VEL
LIN {X 0,Y 230.308,Z 345.532,A -85,B 0,C 180,E1 -20465.433,E2 -20465.433} C_VEL
LIN {X 0,Y 232.516,Z 337.962,A -85,B 0,C 180,E1 -20467.191,E2 -20467.191} C_VEL
LIN {X 0,Y 231.922,Z 330.922,A -85,B 0,C 180,E1 -20468.885,E2 -20468.885} C_VEL
LIN {X 0,Y 230.638,Z 323.132,A -85,B 0,C 180,E1 -20470.574,E2 -20470.574} C_VEL
LIN {X 0,Y 228.72,Z 315.051,A -85,B 0,C 180,E1 -20472.164,E2 -20472.164} C_VEL
LIN {X 0,Y 225.605,Z 305.426,A -85,B 0,C 180,E1 -20473.919,E2 -20473.919} C_VEL
LIN {X 0,Y 222.278,Z 297.675,A -85,B 0,C 180,E1 -20475.281,E2 -20475.281} C_VEL
LIN {X 0,Y 221.077,Z 294.59,A -85,B 0,C 180,E1 -20475.773,E2 -20475.773} C_VEL
LIN {X 0,Y 221.088,Z 292.1,A -85,B 0,C 180,E1 -20479.718,E2 -20479.718} C_VEL
LIN {X 0,Y 220.909,Z 290.446,A -85,B 0,C 180,E1 -20482.815,E2 -20482.815} C_VEL
LIN {X 0,Y 220.804,Z 289.794,A -85,B 0,C 180,E1 -20485.844,E2 -20485.844} C_VEL
LIN {X 0,Y 220.817,Z 289.791,A -85,B 0,C 180,E1 -20489.392,E2 -20489.392} C_VEL
LIN {X 0,Y 220.878,Z 289.782,A -85,B 0,C 180,E1 -20493.552,E2 -20493.552} C_VEL
LIN {X 0,Y 220.85,Z 289.789,A -85,B 0,C 180,E1 -20497.555,E2 -20497.555} C_VEL
LIN {X 0,Y 220.971,Z 289.767,A -85,B 0,C 180,E1 -20502.574,E2 -20502.574} C_VEL
LIN {X 0,Y 221.012,Z 289.767,A -85,B 0,C 180,E1 -20507.142,E2 -20507.142} C_VEL
LIN {X 0,Y 221.186,Z 289.743,A -85,B 0,C 180,E1 -20510.862,E2 -20510.862} C_VEL
LIN {X 0,Y 221.12,Z 289.748,A -85,B 0,C 180,E1 -20514.532,E2 -20514.532} C_VEL
LIN {X 0,Y 221.502,Z 289.699,A -85,B 0,C 180,E1 -20518.185,E2 -20518.185} C_VEL
LIN {X 0,Y 221.503,Z 289.699,A -85,B 0,C 180,E1 -20521.821,E2 -20521.821} C_VEL
LIN {X 0,Y 221.303,Z 289.728,A -85,B 0,C 180,E1 -20527.301,E2 -20527.301} C_VEL
LIN {X 0,Y 221.109,Z 289.755,A -85,B 0,C 180,E1 -20530.997,E2 -20530.997} C_VEL
LIN {X 0,Y 221.01,Z 289.767,A -85,B 0,C 180,E1 -20536.633,E2 -20536.633} C_VEL
LIN {X 0,Y 220.881,Z 289.784,A -85,B 0,C 180,E1 -20540.49,E2 -20540.49} C_VEL
LIN {X 0,Y 220.842,Z 289.793,A -85,B 0,C 180,E1 -20544.441,E2 -20544.441} C_VEL
LIN {X 0,Y 220.799,Z 289.799,A -85,B 0,C 180,E1 -20548.522,E2 -20548.522} C_VEL
LIN {X 0,Y 220.815,Z 289.799,A -85,B 0,C 180,E1 -20552.76,E2 -20552.76} C_VEL
LIN {X 0,Y 220.888,Z 289.978,A -85,B 0,C 180,E1 -20554.189,E2 -20554.189} C_VEL
LIN {X 0,Y 221.269,Z 292.031,A -85,B 0,C 180,E1 -20557.438,E2 -20557.438} C_VEL
LIN {X 0,Y 221.697,Z 295.044,A -85,B 0,C 180,E1 -20561.741,E2 -20561.741} C_VEL
LIN {X 0,Y 222.321,Z 298.819,A -85,B 0,C 180,E1 -20566.645,E2 -20566.645} C_VEL
LIN {X 0,Y 223.045,Z 302.486,A -85,B 0,C 180,E1 -20570.94,E2 -20570.94} C_VEL
LIN {X 0,Y 223.385,Z 304.634,A -85,B 0,C 180,E1 -20573.293,E2 -20573.293} C_VEL
LIN {X 0,Y 223.366,Z 306.767,A -85,B 0,C 180,E1 -20575.507,E2 -20575.507} C_VEL
LIN {X 0,Y 222.635,Z 309.898,A -85,B 0,C 180,E1 -20578.533,E2 -20578.533} C_VEL
LIN {X 0,Y 223.478,Z 313.336,A -85,B 0,C 180,E1 -20578.941,E2 -20578.941} C_VEL
LIN {X 0,Y 225.837,Z 322.125,A -85,B 0,C 180,E1 -20580.141,E2 -20580.141} C_VEL
LIN {X 0,Y 227.824,Z 332.148,A -85,B 0,C 180,E1 -20581.67,E2 -20581.67} C_VEL
LIN {X 0,Y 228.581,Z 337.299,A -85,B 0,C 180,E1 -20582.511,E2 -20582.511} C_VEL
LIN {X 0,Y 228.509,Z 342.299,A -85,B 0,C 180,E1 -20583.297,E2 -20583.297} C_VEL
LIN {X 0,Y 227.333,Z 347.289,A -85,B 0,C 180,E1 -20584.057,E2 -20584.057} C_VEL
LIN {X 0,Y 223.761,Z 356.782,A -85,B 0,C 180,E1 -20585.7,E2 -20585.7} C_VEL
LIN {X 0,Y 222.41,Z 361.209,A -85,B 0,C 180,E1 -20586.694,E2 -20586.694} C_VEL
LIN {X 0,Y 222.162,Z 362.549,A -85,B 0,C 180,E1 -20587.061,E2 -20587.061} C_VEL
LIN {X 0,Y 220.888,Z 367.793,A -85,B 0,C 180,E1 -20588.54,E2 -20588.54} C_VEL
LIN {X 0,Y 218.85,Z 373.205,A -85,B 0,C 180,E1 -20590.297,E2 -20590.297} C_VEL
LIN {X 0,Y 217.059,Z 377.741,A -85,B 0,C 180,E1 -20592.088,E2 -20592.088} C_VEL
LIN {X 0,Y 215.562,Z 381.53,A -85,B 0,C 180,E1 -20593.914,E2 -20593.914} C_VEL
LIN {X 0,Y 213.792,Z 385.882,A -85,B 0,C 180,E1 -20596.699,E2 -20596.699} C_VEL
LIN {X 0,Y 212.904,Z 388.142,A -85,B 0,C 180,E1 -20598.579,E2 -20598.579} C_VEL
LIN {X 0,Y 212.241,Z 389.801,A -85,B 0,C 180,E1 -20600.472,E2 -20600.472} C_VEL
LIN {X 0,Y 211.825,Z 390.914,A -85,B 0,C 180,E1 -20602.376,E2 -20602.376} C_VEL
LIN {X 0,Y 211.521,Z 391.791,A -85,B 0,C 180,E1 -20605.43,E2 -20605.43} C_VEL
LIN {X 0,Y 211.651,Z 391.494,A -85,B 0,C 180,E1 -20608.1,E2 -20608.1} C_VEL
LIN {X 0,Y 211.746,Z 390.613,A -85,B 0,C 180,E1 -20610.002,E2 -20610.002} C_VEL
LIN {X 0,Y 211.722,Z 389.227,A -85,B 0,C 180,E1 -20611.905,E2 -20611.905} C_VEL
LIN {X 0,Y 211.656,Z 385.866,A -85,B 0,C 180,E1 -20615.008,E2 -20615.008} C_VEL
LIN {X 0,Y 211.882,Z 381.758,A -85,B 0,C 180,E1 -20617.627,E2 -20617.627} C_VEL
LIN {X 0,Y 212.321,Z 376.816,A -85,B 0,C 180,E1 -20620.01,E2 -20620.01} C_VEL
LIN {X 0,Y 213.011,Z 370.549,A -85,B 0,C 180,E1 -20622.386,E2 -20622.386} C_VEL
LIN {X 0,Y 213.81,Z 364.422,A -85,B 0,C 180,E1 -20624.275,E2 -20624.275} C_VEL
LIN {X 0,Y 214.759,Z 358.001,A -85,B 0,C 180,E1 -20625.909,E2 -20625.909} C_VEL
LIN {X 0,Y 215.178,Z 352.632,A -85,B 0,C 180,E1 -20627.097,E2 -20627.097} C_VEL
LIN {X 0,Y 215.084,Z 344.447,A -85,B 0,C 180,E1 -20628.624,E2 -20628.624} C_VEL
LIN {X 0,Y 214.877,Z 336.583,A -85,B 0,C 180,E1 -20629.839,E2 -20629.839} C_VEL
LIN {X 0,Y 214.293,Z 327.052,A -85,B 0,C 180,E1 -20631.023,E2 -20631.023} C_VEL
LIN {X 0,Y 213.375,Z 317.5,A -85,B 0,C 180,E1 -20631.949,E2 -20631.949} C_VEL
LIN {X 0,Y 212.509,Z 310.874,A -85,B 0,C 180,E1 -20632.474,E2 -20632.474} C_VEL
LIN {X 0,Y 213.467,Z 305.359,A -85,B 0,C 180,E1 -20637.449,E2 -20637.449} C_VEL
LIN {X 0,Y 214.839,Z 299.619,A -85,B 0,C 180,E1 -20642.67,E2 -20642.67} C_VEL
LIN {X 0,Y 215.018,Z 296.99,A -85,B 0,C 180,E1 -20645.196,E2 -20645.196} C_VEL
LIN {X 0,Y 214.486,Z 293.72,A -85,B 0,C 180,E1 -20648.507,E2 -20648.507} C_VEL
LIN {X 0,Y 213.88,Z 290.657,A -85,B 0,C 180,E1 -20651.874,E2 -20651.874} C_VEL
LIN {X 0,Y 213.718,Z 290.674,A -85,B 0,C 180,E1 -20656.344,E2 -20656.344} C_VEL
LIN {X 0,Y 213.729,Z 290.673,A -85,B 0,C 180,E1 -20659.142,E2 -20659.142} C_VEL
LIN {X 0,Y 213.756,Z 290.671,A -85,B 0,C 180,E1 -20663.711,E2 -20663.711} C_VEL
LIN {X 0,Y 213.808,Z 290.659,A -85,B 0,C 180,E1 -20668.724,E2 -20668.724} C_VEL
LIN {X 0,Y 213.838,Z 290.658,A -85,B 0,C 180,E1 -20672.602,E2 -20672.602} C_VEL
LIN {X 0,Y 213.83,Z 290.658,A -85,B 0,C 180,E1 -20676.972,E2 -20676.972} C_VEL
LIN {X 0,Y 213.902,Z 290.653,A -85,B 0,C 180,E1 -20682.797,E2 -20682.797} C_VEL
LIN {X 0,Y 213.943,Z 290.645,A -85,B 0,C 180,E1 -20686.703,E2 -20686.703} C_VEL
LIN {X 0,Y 214.136,Z 290.62,A -85,B 0,C 180,E1 -20690.552,E2 -20690.552} C_VEL
LIN {X 0,Y 214.105,Z 290.627,A -85,B 0,C 180,E1 -20694.345,E2 -20694.345} C_VEL
LIN {X 0,Y 214.452,Z 290.578,A -85,B 0,C 180,E1 -20698.119,E2 -20698.119} C_VEL
LIN {X 0,Y 214.554,Z 290.564,A -85,B 0,C 180,E1 -20699.997,E2 -20699.997} C_VEL
LIN {X 0,Y 214.453,Z 290.58,A -85,B 0,C 180,E1 -20701.875,E2 -20701.875} C_VEL
LIN {X 0,Y 214.234,Z 290.608,A -85,B 0,C 180,E1 -20707.537,E2 -20707.537} C_VEL
LIN {X 0,Y 214.05,Z 290.626,A -85,B 0,C 180,E1 -20711.358,E2 -20711.358} C_VEL
LIN {X 0,Y 213.936,Z 290.647,A -85,B 0,C 180,E1 -20715.233,E2 -20715.233} C_VEL
LIN {X 0,Y 213.843,Z 290.656,A -85,B 0,C 180,E1 -20719.183,E2 -20719.183} C_VEL
LIN {X 0,Y 213.849,Z 290.653,A -85,B 0,C 180,E1 -20723.223,E2 -20723.223} C_VEL
LIN {X 0,Y 213.83,Z 290.662,A -85,B 0,C 180,E1 -20727.445,E2 -20727.445} C_VEL
LIN {X 0,Y 213.779,Z 290.67,A -85,B 0,C 180,E1 -20731.731,E2 -20731.731} C_VEL
LIN {X 0,Y 213.758,Z 290.669,A -85,B 0,C 180,E1 -20736.281,E2 -20736.281} C_VEL
LIN {X 0,Y 213.826,Z 290.66,A -85,B 0,C 180,E1 -20741.093,E2 -20741.093} C_VEL
LIN {X 0,Y 213.832,Z 290.661,A -85,B 0,C 180,E1 -20743.688,E2 -20743.688} C_VEL
LIN {X 0,Y 213.835,Z 290.659,A -85,B 0,C 180,E1 -20746.352,E2 -20746.352} C_VEL
LIN {X 0,Y 213.815,Z 290.664,A -85,B 0,C 180,E1 -20749.106,E2 -20749.106} C_VEL
LIN {X 0,Y 213.747,Z 290.669,A -85,B 0,C 180,E1 -20753.71,E2 -20753.71} C_VEL
LIN {X 0,Y 213.787,Z 290.667,A -85,B 0,C 180,E1 -20758.72,E2 -20758.72} C_VEL
LIN {X 0,Y 213.816,Z 290.664,A -85,B 0,C 180,E1 -20762.599,E2 -20762.599} C_VEL
LIN {X 0,Y 213.809,Z 290.664,A -85,B 0,C 180,E1 -20766.969,E2 -20766.969} C_VEL
LIN {X 0,Y 213.665,Z 290.68,A -85,B 0,C 180,E1 -20770.794,E2 -20770.794} C_VEL
LIN {X 0,Y 213.593,Z 290.692,A -85,B 0,C 180,E1 -20772.772,E2 -20772.772} C_VEL
LIN {X 0,Y 212.984,Z 290.769,A -85,B 0,C 180,E1 -20778.277,E2 -20778.277} C_VEL
LIN {X 0,Y 212.941,Z 293.467,A -85,B 0,C 180,E1 -20781.727,E2 -20781.727} C_VEL
LIN {X 0,Y 215.291,Z 305.108,A -85,B 0,C 180,E1 -20782.848,E2 -20782.848} C_VEL
LIN {X 0,Y 216.605,Z 314.037,A -85,B 0,C 180,E1 -20783.945,E2 -20783.945} C_VEL
LIN {X 0,Y 217.338,Z 322.031,A -85,B 0,C 180,E1 -20785.128,E2 -20785.128} C_VEL
LIN {X 0,Y 217.03,Z 327.717,A -85,B 0,C 180,E1 -20786.052,E2 -20786.052} C_VEL
LIN {X 0,Y 215.85,Z 335.999,A -85,B 0,C 180,E1 -20787.665,E2 -20787.665} C_VEL
LIN {X 0,Y 214.838,Z 343.657,A -85,B 0,C 180,E1 -20789.529,E2 -20789.529} C_VEL
LIN {X 0,Y 213.916,Z 349.968,A -85,B 0,C 180,E1 -20791.409,E2 -20791.409} C_VEL
LIN {X 0,Y 213.196,Z 355.206,A -85,B 0,C 180,E1 -20793.305,E2 -20793.305} C_VEL
LIN {X 0,Y 212.774,Z 358.602,A -85,B 0,C 180,E1 -20794.734,E2 -20794.734} C_VEL
LIN {X 0,Y 212.294,Z 362.583,A -85,B 0,C 180,E1 -20796.748,E2 -20796.748} C_VEL
LIN {X 0,Y 211.731,Z 366.78,A -85,B 0,C 180,E1 -20799.551,E2 -20799.551} C_VEL
LIN {X 0,Y 211.483,Z 369.005,A -85,B 0,C 180,E1 -20801.499,E2 -20801.499} C_VEL
LIN {X 0,Y 211.461,Z 370.658,A -85,B 0,C 180,E1 -20803.45,E2 -20803.45} C_VEL
LIN {X 0,Y 211.553,Z 371.783,A -85,B 0,C 180,E1 -20805.565,E2 -20805.565} C_VEL
LIN {X 0,Y 211.739,Z 372.23,A -85,B 0,C 180,E1 -20807.378,E2 -20807.378} C_VEL
LIN {X 0,Y 212.138,Z 372.262,A -85,B 0,C 180,E1 -20809.345,E2 -20809.345} C_VEL
LIN {X 0,Y 212.747,Z 371.797,A -85,B 0,C 180,E1 -20811.305,E2 -20811.305} C_VEL
LIN {X 0,Y 213.525,Z 370.807,A -85,B 0,C 180,E1 -20813.261,E2 -20813.261} C_VEL
LIN {X 0,Y 214.975,Z 368.153,A -85,B 0,C 180,E1 -20816.187,E2 -20816.187} C_VEL
LIN {X 0,Y 216.807,Z 364.38,A -85,B 0,C 180,E1 -20818.937,E2 -20818.937} C_VEL
LIN {X 0,Y 218.456,Z 360.645,A -85,B 0,C 180,E1 -20820.977,E2 -20820.977} C_VEL
LIN {X 0,Y 220.612,Z 355.179,A -85,B 0,C 180,E1 -20823.315,E2 -20823.315} C_VEL
LIN {X 0,Y 223.229,Z 348.209,A -85,B 0,C 180,E1 -20825.619,E2 -20825.619} C_VEL
LIN {X 0,Y 225.843,Z 340.189,A -85,B 0,C 180,E1 -20827.637,E2 -20827.637} C_VEL
LIN {X 0,Y 225.708,Z 334.587,A -85,B 0,C 180,E1 -20829.085,E2 -20829.085} C_VEL
LIN {X 0,Y 224.356,Z 325.242,A -85,B 0,C 180,E1 -20831.259,E2 -20831.259} C_VEL
LIN {X 0,Y 222.712,Z 317.871,A -85,B 0,C 180,E1 -20832.824,E2 -20832.824} C_VEL
LIN {X 0,Y 220.204,Z 309.518,A -85,B 0,C 180,E1 -20834.476,E2 -20834.476} C_VEL
LIN {X 0,Y 216.943,Z 301.518,A -85,B 0,C 180,E1 -20836.026,E2 -20836.026} C_VEL
LIN {X 0,Y 215.234,Z 297.902,A -85,B 0,C 180,E1 -20836.714,E2 -20836.714} C_VEL
LIN {X 0,Y 214.087,Z 294.785,A -85,B 0,C 180,E1 -20837.23,E2 -20837.23} C_VEL
LIN {X 0,Y 214.004,Z 292.539,A -85,B 0,C 180,E1 -20841.399,E2 -20841.399} C_VEL
LIN {X 0,Y 213.767,Z 290.673,A -85,B 0,C 180,E1 -20845.273,E2 -20845.273} C_VEL
LIN {X 0,Y 213.765,Z 290.67,A -85,B 0,C 180,E1 -20848.733,E2 -20848.733} C_VEL
LIN {X 0,Y 213.81,Z 290.666,A -85,B 0,C 180,E1 -20852.606,E2 -20852.606} C_VEL
LIN {X 0,Y 213.804,Z 290.664,A -85,B 0,C 180,E1 -20856.976,E2 -20856.976} C_VEL
LIN {X 0,Y 213.93,Z 290.644,A -85,B 0,C 180,E1 -20862.806,E2 -20862.806} C_VEL
LIN {X 0,Y 213.967,Z 290.641,A -85,B 0,C 180,E1 -20866.711,E2 -20866.711} C_VEL
LIN {X 0,Y 214.125,Z 290.621,A -85,B 0,C 180,E1 -20870.558,E2 -20870.558} C_VEL
LIN {X 0,Y 214.081,Z 290.624,A -85,B 0,C 180,E1 -20874.352,E2 -20874.352} C_VEL
LIN {X 0,Y 214.435,Z 290.579,A -85,B 0,C 180,E1 -20878.125,E2 -20878.125} C_VEL
LIN {X 0,Y 214.54,Z 290.574,A -85,B 0,C 180,E1 -20880.003,E2 -20880.003} C_VEL
LIN {X 0,Y 214.436,Z 290.579,A -85,B 0,C 180,E1 -20881.882,E2 -20881.882} C_VEL
LIN {X 0,Y 214.239,Z 290.61,A -85,B 0,C 180,E1 -20887.543,E2 -20887.543} C_VEL
LIN {X 0,Y 214.04,Z 290.635,A -85,B 0,C 180,E1 -20891.365,E2 -20891.365} C_VEL
LIN {X 0,Y 213.927,Z 290.65,A -85,B 0,C 180,E1 -20895.241,E2 -20895.241} C_VEL
LIN {X 0,Y 213.831,Z 290.662,A -85,B 0,C 180,E1 -20899.191,E2 -20899.191} C_VEL
LIN {X 0,Y 213.798,Z 290.669,A -85,B 0,C 180,E1 -20903.236,E2 -20903.236} C_VEL
LIN {X 0,Y 213.782,Z 290.674,A -85,B 0,C 180,E1 -20907.432,E2 -20907.432} C_VEL
LIN {X 0,Y 213.799,Z 290.821,A -85,B 0,C 180,E1 -20912.85,E2 -20912.85} C_VEL
LIN {X 0,Y 214.203,Z 292.805,A -85,B 0,C 180,E1 -20916.201,E2 -20916.201} C_VEL
LIN {X 0,Y 214.704,Z 296.107,A -85,B 0,C 180,E1 -20921.165,E2 -20921.165} C_VEL
LIN {X 0,Y 215.259,Z 299.598,A -85,B 0,C 180,E1 -20925.916,E2 -20925.916} C_VEL
LIN {X 0,Y 216.108,Z 304.035,A -85,B 0,C 180,E1 -20931.31,E2 -20931.31} C_VEL
LIN {X 0,Y 216.402,Z 306.712,A -85,B 0,C 180,E1 -20934.288,E2 -20934.288} C_VEL
LIN {X 0,Y 215.952,Z 309.519,A -85,B 0,C 180,E1 -20937.185,E2 -20937.185} C_VEL
LIN {X 0,Y 216.874,Z 312.977,A -85,B 0,C 180,E1 -20937.633,E2 -20937.633} C_VEL
LIN {X 0,Y 219.714,Z 323.656,A -85,B 0,C 180,E1 -20939.22,E2 -20939.22} C_VEL
LIN {X 0,Y 221.505,Z 333.17,A -85,B 0,C 180,E1 -20940.772,E2 -20940.772} C_VEL
LIN {X 0,Y 222.536,Z 342.434,A -85,B 0,C 180,E1 -20942.453,E2 -20942.453} C_VEL
LIN {X 0,Y 222.933,Z 352.589,A -85,B 0,C 180,E1 -20944.565,E2 -20944.565} C_VEL
LIN {X 0,Y 222.296,Z 361.567,A -85,B 0,C 180,E1 -20946.789,E2 -20946.789} C_VEL
LIN {X 0,Y 222.162,Z 362.549,A -85,B 0,C 180,E1 -20947.061,E2 -20947.061} C_VEL
LIN {X 0,Y 221.39,Z 365.321,A -85,B 0,C 180,E1 -20947.783,E2 -20947.783} C_VEL
LIN {X 0,Y 219.968,Z 367.868,A -85,B 0,C 180,E1 -20948.462,E2 -20948.462} C_VEL
LIN {X 0,Y 216.015,Z 372.681,A -85,B 0,C 180,E1 -20949.784,E2 -20949.784} C_VEL
LIN {X 0,Y 210.951,Z 377.941,A -85,B 0,C 180,E1 -20951.622,E2 -20951.622} C_VEL
LIN {X 0,Y 209.064,Z 380.691,A -85,B 0,C 180,E1 -20952.949,E2 -20952.949} C_VEL
LIN {X 0,Y 207.441,Z 384.549,A -85,B 0,C 180,E1 -20955.283,E2 -20955.283} C_VEL
LIN {X 0,Y 205.934,Z 387.965,A -85,B 0,C 180,E1 -20958.187,E2 -20958.187} C_VEL
LIN {X 0,Y 205.22,Z 389.612,A -85,B 0,C 180,E1 -20960.143,E2 -20960.143} C_VEL
LIN {X 0,Y 204.763,Z 390.671,A -85,B 0,C 180,E1 -20962.112,E2 -20962.112} C_VEL
LIN {X 0,Y 204.446,Z 391.482,A -85,B 0,C 180,E1 -20965.516,E2 -20965.516} C_VEL
LIN {X 0,Y 204.561,Z 391.105,A -85,B 0,C 180,E1 -20968.034,E2 -20968.034} C_VEL
LIN {X 0,Y 204.679,Z 390.196,A -85,B 0,C 180,E1 -20970.003,E2 -20970.003} C_VEL
LIN {X 0,Y 204.633,Z 388.749,A -85,B 0,C 180,E1 -20971.971,E2 -20971.971} C_VEL
LIN {X 0,Y 204.585,Z 385.591,A -85,B 0,C 180,E1 -20974.955,E2 -20974.955} C_VEL
LIN {X 0,Y 204.847,Z 381.096,A -85,B 0,C 180,E1 -20977.89,E2 -20977.89} C_VEL
LIN {X 0,Y 205.284,Z 376.051,A -85,B 0,C 180,E1 -20980.357,E2 -20980.357} C_VEL
LIN {X 0,Y 205.877,Z 371.129,A -85,B 0,C 180,E1 -20982.322,E2 -20982.322} C_VEL
LIN {X 0,Y 206.649,Z 365.181,A -85,B 0,C 180,E1 -20984.277,E2 -20984.277} C_VEL
LIN {X 0,Y 207.759,Z 357.948,A -85,B 0,C 180,E1 -20986.208,E2 -20986.208} C_VEL
LIN {X 0,Y 208.161,Z 352.622,A -85,B 0,C 180,E1 -20987.439,E2 -20987.439} C_VEL
LIN {X 0,Y 208.092,Z 343.411,A -85,B 0,C 180,E1 -20989.198,E2 -20989.198} C_VEL
LIN {X 0,Y 207.848,Z 334.762,A -85,B 0,C 180,E1 -20990.539,E2 -20990.539} C_VEL
LIN {X 0,Y 207.288,Z 326.024,A -85,B 0,C 180,E1 -20991.639,E2 -20991.639} C_VEL
LIN {X 0,Y 206.301,Z 316.616,A -85,B 0,C 180,E1 -20992.575,E2 -20992.575} C_VEL
LIN {X 0,Y 205.519,Z 310.592,A -85,B 0,C 180,E1 -20993.066,E2 -20993.066} C_VEL
LIN {X 0,Y 206.44,Z 305.598,A -85,B 0,C 180,E1 -20997.726,E2 -20997.726} C_VEL
LIN {X 0,Y 207.769,Z 300.268,A -85,B 0,C 180,E1 -21002.769,E2 -21002.769} C_VEL
LIN {X 0,Y 207.957,Z 297.937,A -85,B 0,C 180,E1 -21005.069,E2 -21005.069} C_VEL
LIN {X 0,Y 207.391,Z 294.38,A -85,B 0,C 180,E1 -21008.789,E2 -21008.789} C_VEL
LIN {X 0,Y 206.842,Z 291.534,A -85,B 0,C 180,E1 -21012.143,E2 -21012.143} C_VEL
LIN {X 0,Y 206.637,Z 291.555,A -85,B 0,C 180,E1 -21017.135,E2 -21017.135} C_VEL
LIN {X 0,Y 206.7,Z 291.548,A -85,B 0,C 180,E1 -21021.449,E2 -21021.449} C_VEL
LIN {X 0,Y 206.712,Z 291.547,A -85,B 0,C 180,E1 -21024.688,E2 -21024.688} C_VEL
LIN {X 0,Y 206.736,Z 291.541,A -85,B 0,C 180,E1 -21029.338,E2 -21029.338} C_VEL
LIN {X 0,Y 206.743,Z 291.544,A -85,B 0,C 180,E1 -21033.77,E2 -21033.77} C_VEL
LIN {X 0,Y 206.743,Z 291.536,A -85,B 0,C 180,E1 -21038.038,E2 -21038.038} C_VEL
LIN {X 0,Y 206.835,Z 291.531,A -85,B 0,C 180,E1 -21042.19,E2 -21042.19} C_VEL
LIN {X 0,Y 206.884,Z 291.522,A -85,B 0,C 180,E1 -21046.24,E2 -21046.24} C_VEL
LIN {X 0,Y 207.082,Z 291.498,A -85,B 0,C 180,E1 -21050.227,E2 -21050.227} C_VEL
LIN {X 0,Y 207.065,Z 291.503,A -85,B 0,C 180,E1 -21054.152,E2 -21054.152} C_VEL
LIN {X 0,Y 207.389,Z 291.458,A -85,B 0,C 180,E1 -21058.055,E2 -21058.055} C_VEL
LIN {X 0,Y 207.519,Z 291.44,A -85,B 0,C 180,E1 -21059.997,E2 -21059.997} C_VEL
LIN {X 0,Y 207.39,Z 291.46,A -85,B 0,C 180,E1 -21061.938,E2 -21061.938} C_VEL
LIN {X 0,Y 207.175,Z 291.488,A -85,B 0,C 180,E1 -21067.795,E2 -21067.795} C_VEL
LIN {X 0,Y 206.987,Z 291.507,A -85,B 0,C 180,E1 -21071.751,E2 -21071.751} C_VEL
LIN {X 0,Y 206.87,Z 291.528,A -85,B 0,C 180,E1 -21075.766,E2 -21075.766} C_VEL
LIN {X 0,Y 206.787,Z 291.536,A -85,B 0,C 180,E1 -21079.865,E2 -21079.865} C_VEL
LIN {X 0,Y 206.765,Z 291.54,A -85,B 0,C 180,E1 -21084.068,E2 -21084.068} C_VEL
LIN {X 0,Y 206.744,Z 291.543,A -85,B 0,C 180,E1 -21088.414,E2 -21088.414} C_VEL
LIN {X 0,Y 206.708,Z 291.548,A -85,B 0,C 180,E1 -21092.951,E2 -21092.951} C_VEL
LIN {X 0,Y 206.743,Z 291.545,A -85,B 0,C 180,E1 -21097.721,E2 -21097.721} C_VEL
LIN {X 0,Y 206.75,Z 291.544,A -85,B 0,C 180,E1 -21101.593,E2 -21101.593} C_VEL
LIN {X 0,Y 206.741,Z 291.544,A -85,B 0,C 180,E1 -21105.545,E2 -21105.545} C_VEL
LIN {X 0,Y 206.736,Z 291.543,A -85,B 0,C 180,E1 -21109.763,E2 -21109.763} C_VEL
LIN {X 0,Y 206.724,Z 291.546,A -85,B 0,C 180,E1 -21114.691,E2 -21114.691} C_VEL
LIN {X 0,Y 206.714,Z 291.548,A -85,B 0,C 180,E1 -21119.335,E2 -21119.335} C_VEL
LIN {X 0,Y 206.722,Z 291.546,A -85,B 0,C 180,E1 -21123.768,E2 -21123.768} C_VEL
LIN {X 0,Y 206.703,Z 291.548,A -85,B 0,C 180,E1 -21128.035,E2 -21128.035} C_VEL
LIN {X 0,Y 206.572,Z 291.563,A -85,B 0,C 180,E1 -21132.276,E2 -21132.276} C_VEL
LIN {X 0,Y 206.12,Z 291.619,A -85,B 0,C 180,E1 -21136.189,E2 -21136.189} C_VEL
LIN {X 0,Y 205.928,Z 291.697,A -85,B 0,C 180,E1 -21138.431,E2 -21138.431} C_VEL
LIN {X 0,Y 205.836,Z 293.605,A -85,B 0,C 180,E1 -21141.077,E2 -21141.077} C_VEL
LIN {X 0,Y 208.193,Z 304.913,A -85,B 0,C 180,E1 -21142.237,E2 -21142.237} C_VEL
LIN {X 0,Y 209.495,Z 313.126,A -85,B 0,C 180,E1 -21143.264,E2 -21143.264} C_VEL
LIN {X 0,Y 210.392,Z 322.706,A -85,B 0,C 180,E1 -21144.727,E2 -21144.727} C_VEL
LIN {X 0,Y 210.266,Z 327.047,A -85,B 0,C 180,E1 -21145.444,E2 -21145.444} C_VEL
LIN {X 0,Y 208.856,Z 336.564,A -85,B 0,C 180,E1 -21147.346,E2 -21147.346} C_VEL
LIN {X 0,Y 207.949,Z 343.325,A -85,B 0,C 180,E1 -21149.029,E2 -21149.029} C_VEL
LIN {X 0,Y 206.992,Z 349.743,A -85,B 0,C 180,E1 -21150.97,E2 -21150.97} C_VEL
LIN {X 0,Y 206.212,Z 355.078,A -85,B 0,C 180,E1 -21152.928,E2 -21152.928} C_VEL
LIN {X 0,Y 205.635,Z 359.526,A -85,B 0,C 180,E1 -21154.899,E2 -21154.899} C_VEL
LIN {X 0,Y 205.192,Z 362.932,A -85,B 0,C 180,E1 -21156.69,E2 -21156.69} C_VEL
LIN {X 0,Y 204.737,Z 366.283,A -85,B 0,C 180,E1 -21158.883,E2 -21158.883} C_VEL
LIN {X 0,Y 204.362,Z 369.594,A -85,B 0,C 180,E1 -21161.905,E2 -21161.905} C_VEL
LIN {X 0,Y 204.368,Z 371.176,A -85,B 0,C 180,E1 -21163.926,E2 -21163.926} C_VEL
LIN {X 0,Y 204.489,Z 372.189,A -85,B 0,C 180,E1 -21165.956,E2 -21165.956} C_VEL
LIN {X 0,Y 204.744,Z 372.62,A -85,B 0,C 180,E1 -21167.992,E2 -21167.992} C_VEL
LIN {X 0,Y 205.212,Z 372.551,A -85,B 0,C 180,E1 -21170.025,E2 -21170.025} C_VEL
LIN {X 0,Y 206.381,Z 371.454,A -85,B 0,C 180,E1 -21173.167,E2 -21173.167} C_VEL
LIN {X 0,Y 207.777,Z 369.261,A -85,B 0,C 180,E1 -21176.083,E2 -21176.083} C_VEL
LIN {X 0,Y 209.541,Z 365.955,A -85,B 0,C 180,E1 -21178.822,E2 -21178.822} C_VEL
LIN {X 0,Y 211.28,Z 362.341,A -85,B 0,C 180,E1 -21181.034,E2 -21181.034} C_VEL
LIN {X 0,Y 213.461,Z 357.152,A -85,B 0,C 180,E1 -21183.465,E2 -21183.465} C_VEL
LIN {X 0,Y 215.678,Z 351.73,A -85,B 0,C 180,E1 -21185.456,E2 -21185.456} C_VEL
LIN {X 0,Y 217.856,Z 345.816,A -85,B 0,C 180,E1 -21187.216,E2 -21187.216} C_VEL
LIN {X 0,Y 219.418,Z 340.53,A -85,B 0,C 180,E1 -21188.572,E2 -21188.572} C_VEL
LIN {X 0,Y 218.89,Z 333.015,A -85,B 0,C 180,E1 -21190.582,E2 -21190.582} C_VEL
LIN {X 0,Y 217.714,Z 325.344,A -85,B 0,C 180,E1 -21192.439,E2 -21192.439} C_VEL
LIN {X 0,Y 215.804,Z 317.275,A -85,B 0,C 180,E1 -21194.243,E2 -21194.243} C_VEL
LIN {X 0,Y 213.313,Z 309.398,A -85,B 0,C 180,E1 -21195.899,E2 -21195.899} C_VEL
LIN {X 0,Y 210.222,Z 302.192,A -85,B 0,C 180,E1 -21197.422,E2 -21197.422} C_VEL
LIN {X 0,Y 208.517,Z 298.688,A -85,B 0,C 180,E1 -21198.15,E2 -21198.15} C_VEL
LIN {X 0,Y 207.179,Z 295.545,A -85,B 0,C 180,E1 -21198.758,E2 -21198.758} C_VEL
LIN {X 0,Y 207.126,Z 295.2,A -85,B 0,C 180,E1 -21198.832,E2 -21198.832} C_VEL
LIN {X 0,Y 206.967,Z 293.412,A -85,B 0,C 180,E1 -21202.327,E2 -21202.327} C_VEL
LIN {X 0,Y 206.811,Z 292.263,A -85,B 0,C 180,E1 -21204.716,E2 -21204.716} C_VEL
LIN {X 0,Y 206.689,Z 291.552,A -85,B 0,C 180,E1 -21207.046,E2 -21207.046} C_VEL
LIN {X 0,Y 206.749,Z 291.545,A -85,B 0,C 180,E1 -21212.1,E2 -21212.1} C_VEL
LIN {X 0,Y 206.739,Z 291.542,A -85,B 0,C 180,E1 -21216.607,E2 -21216.607} C_VEL
LIN {X 0,Y 206.859,Z 291.524,A -85,B 0,C 180,E1 -21222.199,E2 -21222.199} C_VEL
LIN {X 0,Y 206.9,Z 291.519,A -85,B 0,C 180,E1 -21226.249,E2 -21226.249} C_VEL
LIN {X 0,Y 207.068,Z 291.498,A -85,B 0,C 180,E1 -21230.233,E2 -21230.233} C_VEL
LIN {X 0,Y 207.043,Z 291.499,A -85,B 0,C 180,E1 -21234.159,E2 -21234.159} C_VEL
LIN {X 0,Y 207.371,Z 291.458,A -85,B 0,C 180,E1 -21238.061,E2 -21238.061} C_VEL
LIN {X 0,Y 207.505,Z 291.451,A -85,B 0,C 180,E1 -21240.003,E2 -21240.003} C_VEL
LIN {X 0,Y 207.373,Z 291.458,A -85,B 0,C 180,E1 -21241.946,E2 -21241.946} C_VEL
LIN {X 0,Y 207.18,Z 291.491,A -85,B 0,C 180,E1 -21247.802,E2 -21247.802} C_VEL
LIN {X 0,Y 206.976,Z 291.516,A -85,B 0,C 180,E1 -21251.759,E2 -21251.759} C_VEL
LIN {X 0,Y 206.861,Z 291.531,A -85,B 0,C 180,E1 -21255.774,E2 -21255.774} C_VEL
LIN {X 0,Y 206.774,Z 291.542,A -85,B 0,C 180,E1 -21259.873,E2 -21259.873} C_VEL
LIN {X 0,Y 206.733,Z 291.548,A -85,B 0,C 180,E1 -21264.079,E2 -21264.079} C_VEL
LIN {X 0,Y 206.684,Z 291.558,A -85,B 0,C 180,E1 -21268.431,E2 -21268.431} C_VEL
LIN {X 0,Y 206.737,Z 291.596,A -85,B 0,C 180,E1 -21271.247,E2 -21271.247} C_VEL
LIN {X 0,Y 207.23,Z 293.984,A -85,B 0,C 180,E1 -21275.523,E2 -21275.523} C_VEL
LIN {X 0,Y 207.631,Z 296.834,A -85,B 0,C 180,E1 -21280.029,E2 -21280.029} C_VEL
LIN {X 0,Y 208.192,Z 300.404,A -85,B 0,C 180,E1 -21285.15,E2 -21285.15} C_VEL
LIN {X 0,Y 208.986,Z 304.709,A -85,B 0,C 180,E1 -21290.67,E2 -21290.67} C_VEL
LIN {X 0,Y 209.367,Z 307.27,A -85,B 0,C 180,E1 -21293.675,E2 -21293.675} C_VEL
LIN {X 0,Y 209.24,Z 309.177,A -85,B 0,C 180,E1 -21295.721,E2 -21295.721} C_VEL
LIN {X 0,Y 210.2,Z 312.537,A -85,B 0,C 180,E1 -21296.194,E2 -21296.194} C_VEL
LIN {X 0,Y 212.614,Z 320.612,A -85,B 0,C 180,E1 -21297.474,E2 -21297.474} C_VEL
LIN {X 0,Y 214.81,Z 331.584,A -85,B 0,C 180,E1 -21299.338,E2 -21299.338} C_VEL
LIN {X 0,Y 215.784,Z 339.235,A -85,B 0,C 180,E1 -21300.758,E2 -21300.758} C_VEL
LIN {X 0,Y 216.319,Z 347.934,A -85,B 0,C 180,E1 -21302.566,E2 -21302.566} C_VEL
LIN {X 0,Y 216.369,Z 354.098,A -85,B 0,C 180,E1 -21303.995,E2 -21303.995} C_VEL
LIN {X 0,Y 215.849,Z 360.867,A -85,B 0,C 180,E1 -21305.743,E2 -21305.743} C_VEL
LIN {X 0,Y 214.797,Z 366.585,A -85,B 0,C 180,E1 -21307.393,E2 -21307.393} C_VEL
LIN {X 0,Y 212.188,Z 373.318,A -85,B 0,C 180,E1 -21309.651,E2 -21309.651} C_VEL
LIN {X 0,Y 210.323,Z 377.773,A -85,B 0,C 180,E1 -21311.494,E2 -21311.494} C_VEL
LIN {X 0,Y 209.064,Z 380.691,A -85,B 0,C 180,E1 -21312.949,E2 -21312.949} C_VEL
LIN {X 0,Y 207.378,Z 383.206,A -85,B 0,C 180,E1 -21314.347,E2 -21314.347} C_VEL
LIN {X 0,Y 203.082,Z 386.536,A -85,B 0,C 180,E1 -21316.667,E2 -21316.667} C_VEL
LIN {X 0,Y 199.747,Z 388.505,A -85,B 0,C 180,E1 -21318.646,E2 -21318.646} C_VEL
LIN {X 0,Y 198.165,Z 389.655,A -85,B 0,C 180,E1 -21320.258,E2 -21320.258} C_VEL
LIN {X 0,Y 197.934,Z 389.924,A -85,B 0,C 180,E1 -21320.819,E2 -21320.819} C_VEL
LIN {X 0,Y 197.427,Z 390.966,A -85,B 0,C 180,E1 -21323.872,E2 -21323.872} C_VEL
LIN {X 0,Y 197.362,Z 391.055,A -85,B 0,C 180,E1 -21325.919,E2 -21325.919} C_VEL
LIN {X 0,Y 197.472,Z 390.695,A -85,B 0,C 180,E1 -21327.963,E2 -21327.963} C_VEL
LIN {X 0,Y 197.613,Z 389.775,A -85,B 0,C 180,E1 -21330.003,E2 -21330.003} C_VEL
LIN {X 0,Y 197.468,Z 387.379,A -85,B 0,C 180,E1 -21333.063,E2 -21333.063} C_VEL
LIN {X 0,Y 197.556,Z 383.629,A -85,B 0,C 180,E1 -21336.129,E2 -21336.129} C_VEL
LIN {X 0,Y 197.961,Z 378.471,A -85,B 0,C 180,E1 -21339.195,E2 -21339.195} C_VEL
LIN {X 0,Y 198.547,Z 372.899,A -85,B 0,C 180,E1 -21341.746,E2 -21341.746} C_VEL
LIN {X 0,Y 199.486,Z 365.898,A -85,B 0,C 180,E1 -21344.28,E2 -21344.28} C_VEL
LIN {X 0,Y 200.767,Z 357.866,A -85,B 0,C 180,E1 -21346.527,E2 -21346.527} C_VEL
LIN {X 0,Y 201.132,Z 351.308,A -85,B 0,C 180,E1 -21348.069,E2 -21348.069} C_VEL
LIN {X 0,Y 201.088,Z 342.744,A -85,B 0,C 180,E1 -21349.745,E2 -21349.745} C_VEL
LIN {X 0,Y 200.91,Z 334.867,A -85,B 0,C 180,E1 -21351.014,E2 -21351.014} C_VEL
LIN {X 0,Y 200.367,Z 326.25,A -85,B 0,C 180,E1 -21352.155,E2 -21352.155} C_VEL
LIN {X 0,Y 199.464,Z 317.201,A -85,B 0,C 180,E1 -21353.109,E2 -21353.109} C_VEL
LIN {X 0,Y 198.543,Z 310.26,A -85,B 0,C 180,E1 -21353.713,E2 -21353.713} C_VEL
LIN {X 0,Y 199.456,Z 305.609,A -85,B 0,C 180,E1 -21358.244,E2 -21358.244} C_VEL
LIN {X 0,Y 200.668,Z 300.966,A -85,B 0,C 180,E1 -21362.797,E2 -21362.797} C_VEL
LIN {X 0,Y 200.922,Z 298.612,A -85,B 0,C 180,E1 -21365.176,E2 -21365.176} C_VEL
LIN {X 0,Y 200.236,Z 294.716,A -85,B 0,C 180,E1 -21369.447,E2 -21369.447} C_VEL
LIN {X 0,Y 199.79,Z 292.412,A -85,B 0,C 180,E1 -21372.209,E2 -21372.209} C_VEL
LIN {X 0,Y 199.592,Z 292.437,A -85,B 0,C 180,E1 -21378.004,E2 -21378.004} C_VEL
LIN {X 0,Y 199.623,Z 292.428,A -85,B 0,C 180,E1 -21380.767,E2 -21380.767} C_VEL
LIN {X 0,Y 199.626,Z 292.432,A -85,B 0,C 180,E1 -21385.713,E2 -21385.713} C_VEL
LIN {X 0,Y 199.713,Z 292.415,A -85,B 0,C 180,E1 -21388.136,E2 -21388.136} C_VEL
LIN {X 0,Y 199.699,Z 292.42,A -85,B 0,C 180,E1 -21392.77,E2 -21392.77} C_VEL
LIN {X 0,Y 199.723,Z 292.413,A -85,B 0,C 180,E1 -21397.224,E2 -21397.224} C_VEL
LIN {X 0,Y 199.76,Z 292.413,A -85,B 0,C 180,E1 -21401.797,E2 -21401.797} C_VEL
LIN {X 0,Y 199.822,Z 292.402,A -85,B 0,C 180,E1 -21405.744,E2 -21405.744} C_VEL
LIN {X 0,Y 200.033,Z 292.375,A -85,B 0,C 180,E1 -21409.879,E2 -21409.879} C_VEL
LIN {X 0,Y 200.027,Z 292.38,A -85,B 0,C 180,E1 -21413.946,E2 -21413.946} C_VEL
LIN {X 0,Y 200.328,Z 292.337,A -85,B 0,C 180,E1 -21417.986,E2 -21417.986} C_VEL
LIN {X 0,Y 200.484,Z 292.316,A -85,B 0,C 180,E1 -21419.996,E2 -21419.996} C_VEL
LIN {X 0,Y 200.039,Z 292.379,A -85,B 0,C 180,E1 -21424.026,E2 -21424.026} C_VEL
LIN {X 0,Y 200.118,Z 292.368,A -85,B 0,C 180,E1 -21428.072,E2 -21428.072} C_VEL
LIN {X 0,Y 199.919,Z 292.389,A -85,B 0,C 180,E1 -21432.173,E2 -21432.173} C_VEL
LIN {X 0,Y 199.808,Z 292.409,A -85,B 0,C 180,E1 -21436.339,E2 -21436.339} C_VEL
LIN {X 0,Y 199.703,Z 292.414,A -85,B 0,C 180,E1 -21440.601,E2 -21440.601} C_VEL
LIN {X 0,Y 199.674,Z 292.422,A -85,B 0,C 180,E1 -21444.98,E2 -21444.98} C_VEL
LIN {X 0,Y 199.675,Z 292.425,A -85,B 0,C 180,E1 -21449.517,E2 -21449.517} C_VEL
LIN {X 0,Y 199.663,Z 292.425,A -85,B 0,C 180,E1 -21452.347,E2 -21452.347} C_VEL
LIN {X 0,Y 199.661,Z 292.425,A -85,B 0,C 180,E1 -21456.749,E2 -21456.749} C_VEL
LIN {X 0,Y 199.721,Z 292.42,A -85,B 0,C 180,E1 -21459.296,E2 -21459.296} C_VEL
LIN {X 0,Y 199.698,Z 292.421,A -85,B 0,C 180,E1 -21462.346,E2 -21462.346} C_VEL
LIN {X 0,Y 199.689,Z 292.423,A -85,B 0,C 180,E1 -21465.257,E2 -21465.257} C_VEL
LIN {X 0,Y 199.691,Z 292.421,A -85,B 0,C 180,E1 -21468.031,E2 -21468.031} C_VEL
LIN {X 0,Y 199.696,Z 292.421,A -85,B 0,C 180,E1 -21470.731,E2 -21470.731} C_VEL
LIN {X 0,Y 199.627,Z 292.43,A -85,B 0,C 180,E1 -21475.713,E2 -21475.713} C_VEL
LIN {X 0,Y 199.695,Z 292.42,A -85,B 0,C 180,E1 -21478.133,E2 -21478.133} C_VEL
LIN {X 0,Y 199.677,Z 292.426,A -85,B 0,C 180,E1 -21482.768,E2 -21482.768} C_VEL
LIN {X 0,Y 199.675,Z 292.424,A -85,B 0,C 180,E1 -21487.219,E2 -21487.219} C_VEL
LIN {X 0,Y 199.533,Z 292.439,A -85,B 0,C 180,E1 -21491.974,E2 -21491.974} C_VEL
LIN {X 0,Y 199.131,Z 292.492,A -85,B 0,C 180,E1 -21495.694,E2 -21495.694} C_VEL
LIN {X 0,Y 198.848,Z 292.593,A -85,B 0,C 180,E1 -21498.53,E2 -21498.53} C_VEL
LIN {X 0,Y 198.782,Z 293.928,A -85,B 0,C 180,E1 -21500.452,E2 -21500.452} C_VEL
LIN {X 0,Y 201.279,Z 305.437,A -85,B 0,C 180,E1 -21501.677,E2 -21501.677} C_VEL
LIN {X 0,Y 202.601,Z 313.797,A -85,B 0,C 180,E1 -21502.774,E2 -21502.774} C_VEL
LIN {X 0,Y 203.394,Z 321.938,A -85,B 0,C 180,E1 -21504.047,E2 -21504.047} C_VEL
LIN {X 0,Y 203.491,Z 326.256,A -85,B 0,C 180,E1 -21504.796,E2 -21504.796} C_VEL
LIN {X 0,Y 202.081,Z 336.077,A -85,B 0,C 180,E1 -21506.758,E2 -21506.758} C_VEL
LIN {X 0,Y 201.094,Z 342.977,A -85,B 0,C 180,E1 -21508.495,E2 -21508.495} C_VEL
LIN {X 0,Y 200.065,Z 349.51,A -85,B 0,C 180,E1 -21510.501,E2 -21510.501} C_VEL
LIN {X 0,Y 199.229,Z 354.942,A -85,B 0,C 180,E1 -21512.525,E2 -21512.525} C_VEL
LIN {X 0,Y 198.486,Z 360.445,A -85,B 0,C 180,E1 -21515.076,E2 -21515.076} C_VEL
LIN {X 0,Y 197.977,Z 363.995,A -85,B 0,C 180,E1 -21517.106,E2 -21517.106} C_VEL
LIN {X 0,Y 197.44,Z 368.168,A -85,B 0,C 180,E1 -21520.249,E2 -21520.249} C_VEL
LIN {X 0,Y 197.252,Z 370.182,A -85,B 0,C 180,E1 -21522.341,E2 -21522.341} C_VEL
LIN {X 0,Y 197.29,Z 371.663,A -85,B 0,C 180,E1 -21524.437,E2 -21524.437} C_VEL
LIN {X 0,Y 197.465,Z 372.634,A -85,B 0,C 180,E1 -21526.54,E2 -21526.54} C_VEL
LIN {X 0,Y 197.772,Z 373.01,A -85,B 0,C 180,E1 -21528.649,E2 -21528.649} C_VEL
LIN {X 0,Y 198.321,Z 372.84,A -85,B 0,C 180,E1 -21530.752,E2 -21530.752} C_VEL
LIN {X 0,Y 199.447,Z 371.809,A -85,B 0,C 180,E1 -21533.639,E2 -21533.639} C_VEL
LIN {X 0,Y 201.164,Z 369.276,A -85,B 0,C 180,E1 -21537.009,E2 -21537.009} C_VEL
LIN {X 0,Y 202.531,Z 366.924,A -85,B 0,C 180,E1 -21539.062,E2 -21539.062} C_VEL
LIN {X 0,Y 204.964,Z 362.076,A -85,B 0,C 180,E1 -21542.102,E2 -21542.102} C_VEL
LIN {X 0,Y 206.83,Z 357.957,A -85,B 0,C 180,E1 -21544.098,E2 -21544.098} C_VEL
LIN {X 0,Y 209.379,Z 352.034,A -85,B 0,C 180,E1 -21546.341,E2 -21546.341} C_VEL
LIN {X 0,Y 211.405,Z 346.841,A -85,B 0,C 180,E1 -21547.95,E2 -21547.95} C_VEL
LIN {X 0,Y 212.952,Z 342.041,A -85,B 0,C 180,E1 -21549.252,E2 -21549.252} C_VEL
LIN {X 0,Y 212.472,Z 334.479,A -85,B 0,C 180,E1 -21551.414,E2 -21551.414} C_VEL
LIN {X 0,Y 211.343,Z 326.527,A -85,B 0,C 180,E1 -21553.449,E2 -21553.449} C_VEL
LIN {X 0,Y 209.265,Z 317.652,A -85,B 0,C 180,E1 -21555.544,E2 -21555.544} C_VEL
LIN {X 0,Y 206.434,Z 309.451,A -85,B 0,C 180,E1 -21557.424,E2 -21557.424} C_VEL
LIN {X 0,Y 203.429,Z 302.777,A -85,B 0,C 180,E1 -21558.98,E2 -21558.98} C_VEL
LIN {X 0,Y 201.787,Z 299.479,A -85,B 0,C 180,E1 -21559.728,E2 -21559.728} C_VEL
LIN {X 0,Y 200.311,Z 296.602,A -85,B 0,C 180,E1 -21560.404,E2 -21560.404} C_VEL
LIN {X 0,Y 200.087,Z 295.619,A -85,B 0,C 180,E1 -21560.596,E2 -21560.596} C_VEL
LIN {X 0,Y 199.753,Z 293.209,A -85,B 0,C 180,E1 -21565.746,E2 -21565.746} C_VEL
LIN {X 0,Y 199.68,Z 292.426,A -85,B 0,C 180,E1 -21568.138,E2 -21568.138} C_VEL
LIN {X 0,Y 199.669,Z 292.426,A -85,B 0,C 180,E1 -21572.774,E2 -21572.774} C_VEL
LIN {X 0,Y 199.7,Z 292.422,A -85,B 0,C 180,E1 -21577.229,E2 -21577.229} C_VEL
LIN {X 0,Y 199.782,Z 292.407,A -85,B 0,C 180,E1 -21581.761,E2 -21581.761} C_VEL
LIN {X 0,Y 199.835,Z 292.398,A -85,B 0,C 180,E1 -21585.752,E2 -21585.752} C_VEL
LIN {X 0,Y 200.01,Z 292.376,A -85,B 0,C 180,E1 -21589.885,E2 -21589.885} C_VEL
LIN {X 0,Y 200.004,Z 292.376,A -85,B 0,C 180,E1 -21593.953,E2 -21593.953} C_VEL
LIN {X 0,Y 200.31,Z 292.337,A -85,B 0,C 180,E1 -21597.993,E2 -21597.993} C_VEL
LIN {X 0,Y 200.469,Z 292.327,A -85,B 0,C 180,E1 -21600.004,E2 -21600.004} C_VEL
LIN {X 0,Y 200.023,Z 292.384,A -85,B 0,C 180,E1 -21604.033,E2 -21604.033} C_VEL
LIN {X 0,Y 200.124,Z 292.371,A -85,B 0,C 180,E1 -21608.079,E2 -21608.079} C_VEL
LIN {X 0,Y 199.908,Z 292.398,A -85,B 0,C 180,E1 -21612.181,E2 -21612.181} C_VEL
LIN {X 0,Y 199.798,Z 292.41,A -85,B 0,C 180,E1 -21616.347,E2 -21616.347} C_VEL
LIN {X 0,Y 199.685,Z 292.424,A -85,B 0,C 180,E1 -21620.61,E2 -21620.61} C_VEL
LIN {X 0,Y 199.646,Z 292.432,A -85,B 0,C 180,E1 -21624.991,E2 -21624.991} C_VEL
LIN {X 0,Y 199.639,Z 292.483,A -85,B 0,C 180,E1 -21629.677,E2 -21629.677} C_VEL
LIN {X 0,Y 200.127,Z 294.789,A -85,B 0,C 180,E1 -21634.19,E2 -21634.19} C_VEL
LIN {X 0,Y 200.624,Z 297.715,A -85,B 0,C 180,E1 -21639.094,E2 -21639.094} C_VEL
LIN {X 0,Y 201.13,Z 301.208,A -85,B 0,C 180,E1 -21644.339,E2 -21644.339} C_VEL
LIN {X 0,Y 201.876,Z 305.39,A -85,B 0,C 180,E1 -21649.991,E2 -21649.991} C_VEL
LIN {X 0,Y 202.351,Z 308.702,A -85,B 0,C 180,E1 -21654.037,E2 -21654.037} C_VEL
LIN {X 0,Y 203.303,Z 311.941,A -85,B 0,C 180,E1 -21654.554,E2 -21654.554} C_VEL
LIN {X 0,Y 204.239,Z 314.117,A -85,B 0,C 180,E1 -21654.991,E2 -21654.991} C_VEL
LIN {X 0,Y 206.794,Z 323.062,A -85,B 0,C 180,E1 -21656.556,E2 -21656.556} C_VEL
LIN {X 0,Y 208.425,Z 331.668,A -85,B 0,C 180,E1 -21658.113,E2 -21658.113} C_VEL
LIN {X 0,Y 209.307,Z 338.146,A -85,B 0,C 180,E1 -21659.375,E2 -21659.375} C_VEL
LIN {X 0,Y 209.864,Z 347.358,A -85,B 0,C 180,E1 -21661.365,E2 -21661.365} C_VEL
LIN {X 0,Y 209.85,Z 354.565,A -85,B 0,C 180,E1 -21663.123,E2 -21663.123} C_VEL
LIN {X 0,Y 209.211,Z 361.755,A -85,B 0,C 180,E1 -21665.1,E2 -21665.1} C_VEL
LIN {X 0,Y 208.25,Z 366.792,A -85,B 0,C 180,E1 -21666.641,E2 -21666.641} C_VEL
LIN {X 0,Y 206.101,Z 372.258,A -85,B 0,C 180,E1 -21668.498,E2 -21668.498} C_VEL
LIN {X 0,Y 203.616,Z 377.804,A -85,B 0,C 180,E1 -21670.861,E2 -21670.861} C_VEL
LIN {X 0,Y 201.184,Z 382.987,A -85,B 0,C 180,E1 -21673.775,E2 -21673.775} C_VEL
LIN {X 0,Y 199.449,Z 386.823,A -85,B 0,C 180,E1 -21676.762,E2 -21676.762} C_VEL
LIN {X 0,Y 198.219,Z 389.406,A -85,B 0,C 180,E1 -21679.792,E2 -21679.792} C_VEL
LIN {X 0,Y 197.934,Z 389.924,A -85,B 0,C 180,E1 -21680.819,E2 -21680.819} C_VEL
LIN {X 0,Y 196.932,Z 390.687,A -85,B 0,C 180,E1 -21682.497,E2 -21682.497} C_VEL
LIN {X 0,Y 193.814,Z 390.949,A -85,B 0,C 180,E1 -21685.254,E2 -21685.254} C_VEL
LIN {X 0,Y 191.009,Z 390.249,A -85,B 0,C 180,E1 -21688.096,E2 -21688.096} C_VEL
LIN {X 0,Y 190.529,Z 389.403,A -85,B 0,C 180,E1 -21689.864,E2 -21689.864} C_VEL
LIN {X 0,Y 190.459,Z 387.781,A -85,B 0,C 180,E1 -21692.117,E2 -21692.117} C_VEL
LIN {X 0,Y 190.435,Z 384.114,A -85,B 0,C 180,E1 -21695.589,E2 -21695.589} C_VEL
LIN {X 0,Y 190.74,Z 379.705,A -85,B 0,C 180,E1 -21698.478,E2 -21698.478} C_VEL
LIN {X 0,Y 191.252,Z 374.489,A -85,B 0,C 180,E1 -21701.126,E2 -21701.126} C_VEL
LIN {X 0,Y 192.172,Z 367.951,A -85,B 0,C 180,E1 -21703.754,E2 -21703.754} C_VEL
LIN {X 0,Y 193.433,Z 359.766,A -85,B 0,C 180,E1 -21706.357,E2 -21706.357} C_VEL
LIN {X 0,Y 194.087,Z 354.662,A -85,B 0,C 180,E1 -21707.656,E2 -21707.656} C_VEL
LIN {X 0,Y 194.165,Z 345.238,A -85,B 0,C 180,E1 -21709.756,E2 -21709.756} C_VEL
LIN {X 0,Y 193.97,Z 335.091,A -85,B 0,C 180,E1 -21711.507,E2 -21711.507} C_VEL
LIN {X 0,Y 193.438,Z 326.091,A -85,B 0,C 180,E1 -21712.753,E2 -21712.753} C_VEL
LIN {X 0,Y 192.465,Z 316.601,A -85,B 0,C 180,E1 -21713.796,E2 -21713.796} C_VEL
LIN {X 0,Y 191.555,Z 309.873,A -85,B 0,C 180,E1 -21714.452,E2 -21714.452} C_VEL
LIN {X 0,Y 192.501,Z 305.584,A -85,B 0,C 180,E1 -21718.806,E2 -21718.806} C_VEL
LIN {X 0,Y 193.702,Z 301.057,A -85,B 0,C 180,E1 -21723.432,E2 -21723.432} C_VEL
LIN {X 0,Y 193.836,Z 299.133,A -85,B 0,C 180,E1 -21725.462,E2 -21725.462} C_VEL
LIN {X 0,Y 193.105,Z 295.053,A -85,B 0,C 180,E1 -21730.152,E2 -21730.152} C_VEL
LIN {X 0,Y 192.719,Z 293.292,A -85,B 0,C 180,E1 -21732.43,E2 -21732.43} C_VEL
LIN {X 0,Y 192.528,Z 293.312,A -85,B 0,C 180,E1 -21736.896,E2 -21736.896} C_VEL
LIN {X 0,Y 192.564,Z 293.308,A -85,B 0,C 180,E1 -21741.647,E2 -21741.647} C_VEL
LIN {X 0,Y 192.612,Z 293.303,A -85,B 0,C 180,E1 -21746.813,E2 -21746.813} C_VEL
LIN {X 0,Y 192.677,Z 293.296,A -85,B 0,C 180,E1 -21751.69,E2 -21751.69} C_VEL
LIN {X 0,Y 192.696,Z 293.289,A -85,B 0,C 180,E1 -21756.344,E2 -21756.344} C_VEL
LIN {X 0,Y 192.708,Z 293.293,A -85,B 0,C 180,E1 -21761.487,E2 -21761.487} C_VEL
LIN {X 0,Y 192.748,Z 293.285,A -85,B 0,C 180,E1 -21765.209,E2 -21765.209} C_VEL
LIN {X 0,Y 192.955,Z 293.257,A -85,B 0,C 180,E1 -21769.564,E2 -21769.564} C_VEL
LIN {X 0,Y 192.989,Z 293.257,A -85,B 0,C 180,E1 -21773.724,E2 -21773.724} C_VEL
LIN {X 0,Y 193.27,Z 293.216,A -85,B 0,C 180,E1 -21777.912,E2 -21777.912} C_VEL
LIN {X 0,Y 193.449,Z 293.192,A -85,B 0,C 180,E1 -21779.996,E2 -21779.996} C_VEL
LIN {X 0,Y 192.985,Z 293.258,A -85,B 0,C 180,E1 -21784.173,E2 -21784.173} C_VEL
LIN {X 0,Y 193.069,Z 293.243,A -85,B 0,C 180,E1 -21788.368,E2 -21788.368} C_VEL
LIN {X 0,Y 192.858,Z 293.271,A -85,B 0,C 180,E1 -21792.626,E2 -21792.626} C_VEL
LIN {X 0,Y 192.761,Z 293.285,A -85,B 0,C 180,E1 -21796.954,E2 -21796.954} C_VEL
LIN {X 0,Y 192.639,Z 293.293,A -85,B 0,C 180,E1 -21801.392,E2 -21801.392} C_VEL
LIN {X 0,Y 192.666,Z 293.296,A -85,B 0,C 180,E1 -21804.22,E2 -21804.22} C_VEL
LIN {X 0,Y 192.65,Z 293.298,A -85,B 0,C 180,E1 -21808.887,E2 -21808.887} C_VEL
LIN {X 0,Y 192.599,Z 293.306,A -85,B 0,C 180,E1 -21813.18,E2 -21813.18} C_VEL
LIN {X 0,Y 192.626,Z 293.302,A -85,B 0,C 180,E1 -21818.328,E2 -21818.328} C_VEL
LIN {X 0,Y 192.63,Z 293.303,A -85,B 0,C 180,E1 -21823.136,E2 -21823.136} C_VEL
LIN {X 0,Y 192.627,Z 293.302,A -85,B 0,C 180,E1 -21826.854,E2 -21826.854} C_VEL
LIN {X 0,Y 192.606,Z 293.305,A -85,B 0,C 180,E1 -21831.658,E2 -21831.658} C_VEL
LIN {X 0,Y 192.592,Z 293.309,A -85,B 0,C 180,E1 -21836.81,E2 -21836.81} C_VEL
LIN {X 0,Y 192.655,Z 293.297,A -85,B 0,C 180,E1 -21841.688,E2 -21841.688} C_VEL
LIN {X 0,Y 192.672,Z 293.298,A -85,B 0,C 180,E1 -21846.341,E2 -21846.341} C_VEL
LIN {X 0,Y 192.477,Z 293.317,A -85,B 0,C 180,E1 -21851.67,E2 -21851.67} C_VEL
LIN {X 0,Y 192.121,Z 293.365,A -85,B 0,C 180,E1 -21855.16,E2 -21855.16} C_VEL
LIN {X 0,Y 191.787,Z 293.49,A -85,B 0,C 180,E1 -21858.638,E2 -21858.638} C_VEL
LIN {X 0,Y 191.749,Z 294.256,A -85,B 0,C 180,E1 -21859.772,E2 -21859.772} C_VEL
LIN {X 0,Y 194.084,Z 304.255,A -85,B 0,C 180,E1 -21860.854,E2 -21860.854} C_VEL
LIN {X 0,Y 195.736,Z 314.536,A -85,B 0,C 180,E1 -21862.259,E2 -21862.259} C_VEL
LIN {X 0,Y 196.48,Z 322.599,A -85,B 0,C 180,E1 -21863.579,E2 -21863.579} C_VEL
LIN {X 0,Y 196.58,Z 326.907,A -85,B 0,C 180,E1 -21864.355,E2 -21864.355} C_VEL
LIN {X 0,Y 195.12,Z 336.626,A -85,B 0,C 180,E1 -21866.383,E2 -21866.383} C_VEL
LIN {X 0,Y 193.941,Z 344.35,A -85,B 0,C 180,E1 -21868.44,E2 -21868.44} C_VEL
LIN {X 0,Y 192.913,Z 350.708,A -85,B 0,C 180,E1 -21870.519,E2 -21870.519} C_VEL
LIN {X 0,Y 192.078,Z 355.992,A -85,B 0,C 180,E1 -21872.619,E2 -21872.619} C_VEL
LIN {X 0,Y 191.319,Z 361.367,A -85,B 0,C 180,E1 -21875.266,E2 -21875.266} C_VEL
LIN {X 0,Y 190.801,Z 364.84,A -85,B 0,C 180,E1 -21877.403,E2 -21877.403} C_VEL
LIN {X 0,Y 190.436,Z 367.675,A -85,B 0,C 180,E1 -21879.557,E2 -21879.557} C_VEL
LIN {X 0,Y 190.162,Z 370.769,A -85,B 0,C 180,E1 -21882.809,E2 -21882.809} C_VEL
LIN {X 0,Y 190.331,Z 372.75,A -85,B 0,C 180,E1 -21886.267,E2 -21886.267} C_VEL
LIN {X 0,Y 190.838,Z 373.384,A -85,B 0,C 180,E1 -21889.353,E2 -21889.353} C_VEL
LIN {X 0,Y 191.482,Z 373.128,A -85,B 0,C 180,E1 -21891.53,E2 -21891.53} C_VEL
LIN {X 0,Y 192.543,Z 372.158,A -85,B 0,C 180,E1 -21894.155,E2 -21894.155} C_VEL
LIN {X 0,Y 194.585,Z 369.256,A -85,B 0,C 180,E1 -21898.001,E2 -21898.001} C_VEL
LIN {X 0,Y 196.782,Z 365.52,A -85,B 0,C 180,E1 -21901.011,E2 -21901.011} C_VEL
LIN {X 0,Y 198.738,Z 361.821,A -85,B 0,C 180,E1 -21903.235,E2 -21903.235} C_VEL
LIN {X 0,Y 200.764,Z 357.57,A -85,B 0,C 180,E1 -21905.279,E2 -21905.279} C_VEL
LIN {X 0,Y 203.466,Z 351.543,A -85,B 0,C 180,E1 -21907.557,E2 -21907.557} C_VEL
LIN {X 0,Y 206.296,Z 344.371,A -85,B 0,C 180,E1 -21909.696,E2 -21909.696} C_VEL
LIN {X 0,Y 206.277,Z 338.679,A -85,B 0,C 180,E1 -21911.455,E2 -21911.455} C_VEL
LIN {X 0,Y 205.604,Z 331.797,A -85,B 0,C 180,E1 -21913.423,E2 -21913.423} C_VEL
LIN {X 0,Y 204.204,Z 323.996,A -85,B 0,C 180,E1 -21915.48,E2 -21915.48} C_VEL
LIN {X 0,Y 202.347,Z 316.949,A -85,B 0,C 180,E1 -21917.239,E2 -21917.239} C_VEL
LIN {X 0,Y 199.273,Z 308.781,A -85,B 0,C 180,E1 -21919.278,E2 -21919.278} C_VEL
LIN {X 0,Y 196.59,Z 303.386,A -85,B 0,C 180,E1 -21920.698,E2 -21920.698} C_VEL
LIN {X 0,Y 194.981,Z 300.235,A -85,B 0,C 180,E1 -21921.485,E2 -21921.485} C_VEL
LIN {X 0,Y 193.317,Z 297.427,A -85,B 0,C 180,E1 -21922.272,E2 -21922.272} C_VEL
LIN {X 0,Y 192.94,Z 296.052,A -85,B 0,C 180,E1 -21922.514,E2 -21922.514} C_VEL
LIN {X 0,Y 192.716,Z 294.103,A -85,B 0,C 180,E1 -21927.005,E2 -21927.005} C_VEL
LIN {X 0,Y 192.583,Z 293.307,A -85,B 0,C 180,E1 -21929.281,E2 -21929.281} C_VEL
LIN {X 0,Y 192.645,Z 293.3,A -85,B 0,C 180,E1 -21931.694,E2 -21931.694} C_VEL
LIN {X 0,Y 192.67,Z 293.294,A -85,B 0,C 180,E1 -21936.349,E2 -21936.349} C_VEL
LIN {X 0,Y 192.718,Z 293.288,A -85,B 0,C 180,E1 -21941.461,E2 -21941.461} C_VEL
LIN {X 0,Y 192.759,Z 293.281,A -85,B 0,C 180,E1 -21945.218,E2 -21945.218} C_VEL
LIN {X 0,Y 192.933,Z 293.257,A -85,B 0,C 180,E1 -21949.57,E2 -21949.57} C_VEL
LIN {X 0,Y 192.966,Z 293.252,A -85,B 0,C 180,E1 -21953.731,E2 -21953.731} C_VEL
LIN {X 0,Y 193.252,Z 293.216,A -85,B 0,C 180,E1 -21957.92,E2 -21957.92} C_VEL
LIN {X 0,Y 193.433,Z 293.204,A -85,B 0,C 180,E1 -21960.004,E2 -21960.004} C_VEL
LIN {X 0,Y 192.97,Z 293.262,A -85,B 0,C 180,E1 -21964.181,E2 -21964.181} C_VEL
LIN {X 0,Y 193.071,Z 293.25,A -85,B 0,C 180,E1 -21968.376,E2 -21968.376} C_VEL
LIN {X 0,Y 192.847,Z 293.276,A -85,B 0,C 180,E1 -21972.634,E2 -21972.634} C_VEL
LIN {X 0,Y 192.751,Z 293.287,A -85,B 0,C 180,E1 -21976.963,E2 -21976.963} C_VEL
LIN {X 0,Y 192.615,Z 293.307,A -85,B 0,C 180,E1 -21981.403,E2 -21981.403} C_VEL
LIN {X 0,Y 192.635,Z 293.305,A -85,B 0,C 180,E1 -21984.212,E2 -21984.212} C_VEL
LIN {X 0,Y 192.643,Z 293.516,A -85,B 0,C 180,E1 -21988.315,E2 -21988.315} C_VEL
LIN {X 0,Y 193.076,Z 295.82,A -85,B 0,C 180,E1 -21993.16,E2 -21993.16} C_VEL
LIN {X 0,Y 193.465,Z 297.904,A -85,B 0,C 180,E1 -21996.952,E2 -21996.952} C_VEL
LIN {X 0,Y 193.765,Z 300.226,A -85,B 0,C 180,E1 -22000.763,E2 -22000.763} C_VEL
LIN {X 0,Y 194.086,Z 302.056,A -85,B 0,C 180,E1 -22003.601,E2 -22003.601} C_VEL
LIN {X 0,Y 194.765,Z 306.083,A -85,B 0,C 180,E1 -22009.273,E2 -22009.273} C_VEL
LIN {X 0,Y 195.151,Z 308.284,A -85,B 0,C 180,E1 -22012.144,E2 -22012.144} C_VEL
LIN {X 0,Y 196.255,Z 311.384,A -85,B 0,C 180,E1 -22012.711,E2 -22012.711} C_VEL
LIN {X 0,Y 197.524,Z 313.902,A -85,B 0,C 180,E1 -22013.307,E2 -22013.307} C_VEL
LIN {X 0,Y 199.645,Z 319.779,A -85,B 0,C 180,E1 -22014.472,E2 -22014.472} C_VEL
LIN {X 0,Y 201.686,Z 329.103,A -85,B 0,C 180,E1 -22016.261,E2 -22016.261} C_VEL
LIN {X 0,Y 203.043,Z 339.086,A -85,B 0,C 180,E1 -22018.335,E2 -22018.335} C_VEL
LIN {X 0,Y 203.456,Z 346.577,A -85,B 0,C 180,E1 -22020.027,E2 -22020.027} C_VEL
LIN {X 0,Y 203.451,Z 353.068,A -85,B 0,C 180,E1 -22021.645,E2 -22021.645} C_VEL
LIN {X 0,Y 202.917,Z 360.258,A -85,B 0,C 180,E1 -22023.665,E2 -22023.665} C_VEL
LIN {X 0,Y 201.709,Z 367.015,A -85,B 0,C 180,E1 -22025.836,E2 -22025.836} C_VEL
LIN {X 0,Y 199.531,Z 372.38,A -85,B 0,C 180,E1 -22027.753,E2 -22027.753} C_VEL
LIN {X 0,Y 196.938,Z 377.84,A -85,B 0,C 180,E1 -22030.186,E2 -22030.186} C_VEL
LIN {X 0,Y 194.362,Z 382.945,A -85,B 0,C 180,E1 -22033.188,E2 -22033.188} C_VEL
LIN {X 0,Y 192.519,Z 386.708,A -85,B 0,C 180,E1 -22036.277,E2 -22036.277} C_VEL
LIN {X 0,Y 191.237,Z 389.181,A -85,B 0,C 180,E1 -22039.415,E2 -22039.415} C_VEL
LIN {X 0,Y 190.692,Z 390.192,A -85,B 0,C 180,E1 -22041.525,E2 -22041.525} C_VEL
LIN {X 0,Y 190.368,Z 390.665,A -85,B 0,C 180,E1 -22043.644,E2 -22043.644} C_VEL
LIN {X 0,Y 190.284,Z 390.694,A -85,B 0,C 180,E1 -22045.767,E2 -22045.767} C_VEL
LIN {X 0,Y 190.387,Z 390.273,A -85,B 0,C 180,E1 -22047.887,E2 -22047.887} C_VEL
LIN {X 0,Y 190.529,Z 389.403,A -85,B 0,C 180,E1 -22049.864,E2 -22049.864} C_VEL
LIN {X 0,Y 190.317,Z 388.752,A -85,B 0,C 180,E1 -22051.025,E2 -22051.025} C_VEL
LIN {X 0,Y 189.541,Z 387.87,A -85,B 0,C 180,E1 -22052.157,E2 -22052.157} C_VEL
LIN {X 0,Y 187.094,Z 385.556,A -85,B 0,C 180,E1 -22054.35,E2 -22054.35} C_VEL
LIN {X 0,Y 184.629,Z 382.587,A -85,B 0,C 180,E1 -22056.54,E2 -22056.54} C_VEL
LIN {X 0,Y 183.693,Z 380.064,A -85,B 0,C 180,E1 -22058.204,E2 -22058.204} C_VEL
LIN {X 0,Y 183.688,Z 379.085,A -85,B 0,C 180,E1 -22058.759,E2 -22058.759} C_VEL
LIN {X 0,Y 184.125,Z 374.895,A -85,B 0,C 180,E1 -22061.005,E2 -22061.005} C_VEL
LIN {X 0,Y 184.812,Z 369.939,A -85,B 0,C 180,E1 -22063.192,E2 -22063.192} C_VEL
LIN {X 0,Y 185.703,Z 363.949,A -85,B 0,C 180,E1 -22065.365,E2 -22065.365} C_VEL
LIN {X 0,Y 186.979,Z 356.671,A -85,B 0,C 180,E1 -22067.502,E2 -22067.502} C_VEL
LIN {X 0,Y 187.156,Z 349.949,A -85,B 0,C 180,E1 -22069.185,E2 -22069.185} C_VEL
LIN {X 0,Y 187.174,Z 341.51,A -85,B 0,C 180,E1 -22070.938,E2 -22070.938} C_VEL
LIN {X 0,Y 186.98,Z 333.529,A -85,B 0,C 180,E1 -22072.305,E2 -22072.305} C_VEL
LIN {X 0,Y 186.408,Z 324.259,A -85,B 0,C 180,E1 -22073.597,E2 -22073.597} C_VEL
LIN {X 0,Y 185.272,Z 314.663,A -85,B 0,C 180,E1 -22074.665,E2 -22074.665} C_VEL
LIN {X 0,Y 184.592,Z 309.61,A -85,B 0,C 180,E1 -22075.138,E2 -22075.138} C_VEL
LIN {X 0,Y 185.891,Z 304.366,A -85,B 0,C 180,E1 -22080.693,E2 -22080.693} C_VEL
LIN {X 0,Y 186.662,Z 301.201,A -85,B 0,C 180,E1 -22084.068,E2 -22084.068} C_VEL
LIN {X 0,Y 186.743,Z 299.735,A -85,B 0,C 180,E1 -22085.689,E2 -22085.689} C_VEL
LIN {X 0,Y 186.121,Z 296.184,A -85,B 0,C 180,E1 -22089.939,E2 -22089.939} C_VEL
LIN {X 0,Y 185.659,Z 294.171,A -85,B 0,C 180,E1 -22092.679,E2 -22092.679} C_VEL
LIN {X 0,Y 185.492,Z 294.189,A -85,B 0,C 180,E1 -22096.996,E2 -22096.996} C_VEL
LIN {X 0,Y 185.481,Z 294.193,A -85,B 0,C 180,E1 -22099.894,E2 -22099.894} C_VEL
LIN {X 0,Y 185.519,Z 294.184,A -85,B 0,C 180,E1 -22102.711,E2 -22102.711} C_VEL
LIN {X 0,Y 185.559,Z 294.178,A -85,B 0,C 180,E1 -22107.974,E2 -22107.974} C_VEL
LIN {X 0,Y 185.595,Z 294.174,A -85,B 0,C 180,E1 -22110.574,E2 -22110.574} C_VEL
LIN {X 0,Y 185.592,Z 294.177,A -85,B 0,C 180,E1 -22115.379,E2 -22115.379} C_VEL
LIN {X 0,Y 185.639,Z 294.173,A -85,B 0,C 180,E1 -22121.174,E2 -22121.174} C_VEL
LIN {X 0,Y 185.678,Z 294.168,A -85,B 0,C 180,E1 -22124.632,E2 -22124.632} C_VEL
LIN {X 0,Y 185.898,Z 294.137,A -85,B 0,C 180,E1 -22129.416,E2 -22129.416} C_VEL
LIN {X 0,Y 185.951,Z 294.134,A -85,B 0,C 180,E1 -22133.486,E2 -22133.486} C_VEL
LIN {X 0,Y 186.214,Z 294.094,A -85,B 0,C 180,E1 -22137.833,E2 -22137.833} C_VEL
LIN {X 0,Y 186.412,Z 294.068,A -85,B 0,C 180,E1 -22139.996,E2 -22139.996} C_VEL
LIN {X 0,Y 185.933,Z 294.138,A -85,B 0,C 180,E1 -22144.332,E2 -22144.332} C_VEL
LIN {X 0,Y 186.016,Z 294.119,A -85,B 0,C 180,E1 -22148.688,E2 -22148.688} C_VEL
LIN {X 0,Y 185.769,Z 294.153,A -85,B 0,C 180,E1 -22153.116,E2 -22153.116} C_VEL
LIN {X 0,Y 185.678,Z 294.165,A -85,B 0,C 180,E1 -22158.862,E2 -22158.862} C_VEL
LIN {X 0,Y 185.603,Z 294.175,A -85,B 0,C 180,E1 -22164.657,E2 -22164.657} C_VEL
LIN {X 0,Y 185.579,Z 294.181,A -85,B 0,C 180,E1 -22169.488,E2 -22169.488} C_VEL
LIN {X 0,Y 185.521,Z 294.186,A -85,B 0,C 180,E1 -22174.622,E2 -22174.622} C_VEL
LIN {X 0,Y 185.566,Z 294.183,A -85,B 0,C 180,E1 -22177.309,E2 -22177.309} C_VEL
LIN {X 0,Y 185.592,Z 294.176,A -85,B 0,C 180,E1 -22180.764,E2 -22180.764} C_VEL
LIN {X 0,Y 185.582,Z 294.178,A -85,B 0,C 180,E1 -22186.009,E2 -22186.009} C_VEL
LIN {X 0,Y 185.56,Z 294.18,A -85,B 0,C 180,E1 -22189.916,E2 -22189.916} C_VEL
LIN {X 0,Y 185.569,Z 294.182,A -85,B 0,C 180,E1 -22192.699,E2 -22192.699} C_VEL
LIN {X 0,Y 185.537,Z 294.183,A -85,B 0,C 180,E1 -22197.971,E2 -22197.971} C_VEL
LIN {X 0,Y 185.573,Z 294.182,A -85,B 0,C 180,E1 -22200.571,E2 -22200.571} C_VEL
LIN {X 0,Y 185.57,Z 294.181,A -85,B 0,C 180,E1 -22205.377,E2 -22205.377} C_VEL
LIN {X 0,Y 185.43,Z 294.2,A -85,B 0,C 180,E1 -22210.053,E2 -22210.053} C_VEL
LIN {X 0,Y 185.39,Z 294.201,A -85,B 0,C 180,E1 -22212.343,E2 -22212.343} C_VEL
LIN {X 0,Y 184.772,Z 294.277,A -85,B 0,C 180,E1 -22218.478,E2 -22218.478} C_VEL
LIN {X 0,Y 184.734,Z 294.587,A -85,B 0,C 180,E1 -22219.032,E2 -22219.032} C_VEL
LIN {X 0,Y 187.11,Z 304.255,A -85,B 0,C 180,E1 -22220.137,E2 -22220.137} C_VEL
LIN {X 0,Y 188.876,Z 315.234,A -85,B 0,C 180,E1 -22221.707,E2 -22221.707} C_VEL
LIN {X 0,Y 189.59,Z 323.232,A -85,B 0,C 180,E1 -22223.078,E2 -22223.078} C_VEL
LIN {X 0,Y 189.694,Z 327.527,A -85,B 0,C 180,E1 -22223.883,E2 -22223.883} C_VEL
LIN {X 0,Y 188.168,Z 337.163,A -85,B 0,C 180,E1 -22225.982,E2 -22225.982} C_VEL
LIN {X 0,Y 187.094,Z 343.995,A -85,B 0,C 180,E1 -22227.844,E2 -22227.844} C_VEL
LIN {X 0,Y 185.984,Z 350.47,A -85,B 0,C 180,E1 -22229.997,E2 -22229.997} C_VEL
LIN {X 0,Y 185.113,Z 355.849,A -85,B 0,C 180,E1 -22232.173,E2 -22232.173} C_VEL
LIN {X 0,Y 184.429,Z 360.341,A -85,B 0,C 180,E1 -22234.368,E2 -22234.368} C_VEL
LIN {X 0,Y 183.885,Z 364.087,A -85,B 0,C 180,E1 -22236.581,E2 -22236.581} C_VEL
LIN {X 0,Y 183.458,Z 367.157,A -85,B 0,C 180,E1 -22238.811,E2 -22238.811} C_VEL
LIN {X 0,Y 183.171,Z 369.551,A -85,B 0,C 180,E1 -22241.057,E2 -22241.057} C_VEL
LIN {X 0,Y 183.061,Z 371.355,A -85,B 0,C 180,E1 -22243.315,E2 -22243.315} C_VEL
LIN {X 0,Y 183.277,Z 373.076,A -85,B 0,C 180,E1 -22246.551,E2 -22246.551} C_VEL
LIN {X 0,Y 183.933,Z 373.71,A -85,B 0,C 180,E1 -22250.111,E2 -22250.111} C_VEL
LIN {X 0,Y 184.662,Z 373.418,A -85,B 0,C 180,E1 -22252.367,E2 -22252.367} C_VEL
LIN {X 0,Y 185.674,Z 372.505,A -85,B 0,C 180,E1 -22254.722,E2 -22254.722} C_VEL
LIN {X 0,Y 186.743,Z 371.171,A -85,B 0,C 180,E1 -22256.844,E2 -22256.844} C_VEL
LIN {X 0,Y 188.891,Z 368.07,A -85,B 0,C 180,E1 -22260.148,E2 -22260.148} C_VEL
LIN {X 0,Y 191.574,Z 363.529,A -85,B 0,C 180,E1 -22263.383,E2 -22263.383} C_VEL
LIN {X 0,Y 194.189,Z 358.39,A -85,B 0,C 180,E1 -22266.019,E2 -22266.019} C_VEL
LIN {X 0,Y 196.872,Z 352.778,A -85,B 0,C 180,E1 -22268.253,E2 -22268.253} C_VEL
LIN {X 0,Y 199.261,Z 347.171,A -85,B 0,C 180,E1 -22270.063,E2 -22270.063} C_VEL
LIN {X 0,Y 199.867,Z 345.403,A -85,B 0,C 180,E1 -22270.577,E2 -22270.577} C_VEL
LIN {X 0,Y 199.873,Z 339.84,A -85,B 0,C 180,E1 -22272.411,E2 -22272.411} C_VEL
LIN {X 0,Y 199.289,Z 333.192,A -85,B 0,C 180,E1 -22274.436,E2 -22274.436} C_VEL
LIN {X 0,Y 198.087,Z 325.927,A -85,B 0,C 180,E1 -22276.489,E2 -22276.489} C_VEL
LIN {X 0,Y 196.138,Z 318.612,A -85,B 0,C 180,E1 -22278.487,E2 -22278.487} C_VEL
LIN {X 0,Y 193.352,Z 311.289,A -85,B 0,C 180,E1 -22280.505,E2 -22280.505} C_VEL
LIN {X 0,Y 190.916,Z 305.746,A -85,B 0,C 180,E1 -22282.04,E2 -22282.04} C_VEL
LIN {X 0,Y 188.82,Z 302.17,A -85,B 0,C 180,E1 -22283.104,E2 -22283.104} C_VEL
LIN {X 0,Y 187.654,Z 300.296,A -85,B 0,C 180,E1 -22283.692,E2 -22283.692} C_VEL
LIN {X 0,Y 186.037,Z 297.178,A -85,B 0,C 180,E1 -22284.58,E2 -22284.58} C_VEL
LIN {X 0,Y 185.867,Z 296.455,A -85,B 0,C 180,E1 -22284.792,E2 -22284.792} C_VEL
LIN {X 0,Y 185.675,Z 295.206,A -85,B 0,C 180,E1 -22288.006,E2 -22288.006} C_VEL
LIN {X 0,Y 185.565,Z 294.244,A -85,B 0,C 180,E1 -22290.579,E2 -22290.579} C_VEL
LIN {X 0,Y 185.565,Z 294.181,A -85,B 0,C 180,E1 -22295.384,E2 -22295.384} C_VEL
LIN {X 0,Y 185.66,Z 294.17,A -85,B 0,C 180,E1 -22301.137,E2 -22301.137} C_VEL
LIN {X 0,Y 185.711,Z 294.163,A -85,B 0,C 180,E1 -22304.643,E2 -22304.643} C_VEL
LIN {X 0,Y 185.876,Z 294.136,A -85,B 0,C 180,E1 -22309.422,E2 -22309.422} C_VEL
LIN {X 0,Y 185.93,Z 294.128,A -85,B 0,C 180,E1 -22313.493,E2 -22313.493} C_VEL
LIN {X 0,Y 186.195,Z 294.095,A -85,B 0,C 180,E1 -22317.841,E2 -22317.841} C_VEL
LIN {X 0,Y 186.397,Z 294.08,A -85,B 0,C 180,E1 -22320.004,E2 -22320.004} C_VEL
LIN {X 0,Y 185.918,Z 294.14,A -85,B 0,C 180,E1 -22324.34,E2 -22324.34} C_VEL
LIN {X 0,Y 186.021,Z 294.126,A -85,B 0,C 180,E1 -22328.696,E2 -22328.696} C_VEL
LIN {X 0,Y 185.758,Z 294.158,A -85,B 0,C 180,E1 -22333.125,E2 -22333.125} C_VEL
LIN {X 0,Y 185.684,Z 294.169,A -85,B 0,C 180,E1 -22337.629,E2 -22337.629} C_VEL
LIN {X 0,Y 185.572,Z 294.183,A -85,B 0,C 180,E1 -22342.258,E2 -22342.258} C_VEL
LIN {X 0,Y 185.573,Z 294.187,A -85,B 0,C 180,E1 -22344.65,E2 -22344.65} C_VEL
LIN {X 0,Y 185.579,Z 294.649,A -85,B 0,C 180,E1 -22347.033,E2 -22347.033} C_VEL
LIN {X 0,Y 186.04,Z 296.832,A -85,B 0,C 180,E1 -22351.933,E2 -22351.933} C_VEL
LIN {X 0,Y 186.552,Z 299.477,A -85,B 0,C 180,E1 -22357.073,E2 -22357.073} C_VEL
LIN {X 0,Y 186.979,Z 302.781,A -85,B 0,C 180,E1 -22362.58,E2 -22362.58} C_VEL
LIN {X 0,Y 187.512,Z 306.094,A -85,B 0,C 180,E1 -22367.578,E2 -22367.578} C_VEL
LIN {X 0,Y 187.873,Z 307.828,A -85,B 0,C 180,E1 -22369.976,E2 -22369.976} C_VEL
LIN {X 0,Y 188.92,Z 310.803,A -85,B 0,C 180,E1 -22370.574,E2 -22370.574} C_VEL
LIN {X 0,Y 190.621,Z 313.752,A -85,B 0,C 180,E1 -22371.407,E2 -22371.407} C_VEL
LIN {X 0,Y 192.534,Z 317.925,A -85,B 0,C 180,E1 -22372.402,E2 -22372.402} C_VEL
LIN {X 0,Y 194.605,Z 324.78,A -85,B 0,C 180,E1 -22373.912,E2 -22373.912} C_VEL
LIN {X 0,Y 196.381,Z 335.081,A -85,B 0,C 180,E1 -22376.084,E2 -22376.084} C_VEL
LIN {X 0,Y 197.125,Z 345.896,A -85,B 0,C 180,E1 -22378.62,E2 -22378.62} C_VEL
LIN {X 0,Y 197.028,Z 353.558,A -85,B 0,C 180,E1 -22380.632,E2 -22380.632} C_VEL
LIN {X 0,Y 196.416,Z 360.898,A -85,B 0,C 180,E1 -22382.824,E2 -22382.824} C_VEL
LIN {X 0,Y 195.189,Z 367.246,A -85,B 0,C 180,E1 -22384.975,E2 -22384.975} C_VEL
LIN {X 0,Y 192.997,Z 372.51,A -85,B 0,C 180,E1 -22386.958,E2 -22386.958} C_VEL
LIN {X 0,Y 190.273,Z 377.885,A -85,B 0,C 180,E1 -22389.461,E2 -22389.461} C_VEL
LIN {X 0,Y 188.4,Z 381.384,A -85,B 0,C 180,E1 -22391.517,E2 -22391.517} C_VEL
LIN {X 0,Y 186.215,Z 385.438,A -85,B 0,C 180,E1 -22394.684,E2 -22394.684} C_VEL
LIN {X 0,Y 185.087,Z 387.435,A -85,B 0,C 180,E1 -22396.834,E2 -22396.834} C_VEL
LIN {X 0,Y 184.238,Z 388.944,A -85,B 0,C 180,E1 -22399.008,E2 -22399.008} C_VEL
LIN {X 0,Y 183.664,Z 389.943,A -85,B 0,C 180,E1 -22401.199,E2 -22401.199} C_VEL
LIN {X 0,Y 183.31,Z 390.365,A -85,B 0,C 180,E1 -22403.398,E2 -22403.398} C_VEL
LIN {X 0,Y 183.193,Z 390.289,A -85,B 0,C 180,E1 -22405.957,E2 -22405.957} C_VEL
LIN {X 0,Y 183.304,Z 389.851,A -85,B 0,C 180,E1 -22407.806,E2 -22407.806} C_VEL
LIN {X 0,Y 183.482,Z 388.89,A -85,B 0,C 180,E1 -22410.003,E2 -22410.003} C_VEL
LIN {X 0,Y 183.287,Z 386.217,A -85,B 0,C 180,E1 -22413.361,E2 -22413.361} C_VEL
LIN {X 0,Y 183.355,Z 384.05,A -85,B 0,C 180,E1 -22415.391,E2 -22415.391} C_VEL
LIN {X 0,Y 183.688,Z 379.085,A -85,B 0,C 180,E1 -22418.759,E2 -22418.759} C_VEL
LIN {X 0,Y 183.321,Z 376.254,A -85,B 0,C 180,E1 -22420.361,E2 -22420.361} C_VEL
LIN {X 0,Y 181.124,Z 370.909,A -85,B 0,C 180,E1 -22422.892,E2 -22422.892} C_VEL
LIN {X 0,Y 179.182,Z 364.859,A -85,B 0,C 180,E1 -22425.317,E2 -22425.317} C_VEL
LIN {X 0,Y 179.24,Z 360.677,A -85,B 0,C 180,E1 -22426.707,E2 -22426.707} C_VEL
LIN {X 0,Y 180.037,Z 355.507,A -85,B 0,C 180,E1 -22428.2,E2 -22428.2} C_VEL
LIN {X 0,Y 180.212,Z 347.206,A -85,B 0,C 180,E1 -22430.278,E2 -22430.278} C_VEL
LIN {X 0,Y 180.193,Z 336.958,A -85,B 0,C 180,E1 -22432.353,E2 -22432.353} C_VEL
LIN {X 0,Y 179.713,Z 326.676,A -85,B 0,C 180,E1 -22433.956,E2 -22433.956} C_VEL
LIN {X 0,Y 178.651,Z 316.592,A -85,B 0,C 180,E1 -22435.196,E2 -22435.196} C_VEL
LIN {X 0,Y 177.681,Z 309.297,A -85,B 0,C 180,E1 -22435.952,E2 -22435.952} C_VEL
LIN {X 0,Y 179.119,Z 303.824,A -85,B 0,C 180,E1 -22441.988,E2 -22441.988} C_VEL
LIN {X 0,Y 179.624,Z 301.356,A -85,B 0,C 180,E1 -22444.744,E2 -22444.744} C_VEL
LIN {X 0,Y 179.661,Z 300.354,A -85,B 0,C 180,E1 -22445.931,E2 -22445.931} C_VEL
LIN {X 0,Y 179.02,Z 296.888,A -85,B 0,C 180,E1 -22450.256,E2 -22450.256} C_VEL
LIN {X 0,Y 178.64,Z 295.046,A -85,B 0,C 180,E1 -22452.668,E2 -22452.668} C_VEL
LIN {X 0,Y 178.421,Z 295.072,A -85,B 0,C 180,E1 -22458.457,E2 -22458.457} C_VEL
LIN {X 0,Y 178.435,Z 295.07,A -85,B 0,C 180,E1 -22463.782,E2 -22463.782} C_VEL
LIN {X 0,Y 178.5,Z 295.061,A -85,B 0,C 180,E1 -22466.545,E2 -22466.545} C_VEL
LIN {X 0,Y 178.536,Z 295.053,A -85,B 0,C 180,E1 -22470.005,E2 -22470.005} C_VEL
LIN {X 0,Y 178.532,Z 295.057,A -85,B 0,C 180,E1 -22474.884,E2 -22474.884} C_VEL
LIN {X 0,Y 178.621,Z 295.047,A -85,B 0,C 180,E1 -22481.649,E2 -22481.649} C_VEL
LIN {X 0,Y 178.653,Z 295.039,A -85,B 0,C 180,E1 -22486.344,E2 -22486.344} C_VEL
LIN {X 0,Y 178.916,Z 295.009,A -85,B 0,C 180,E1 -22490.956,E2 -22490.956} C_VEL
LIN {X 0,Y 179.159,Z 294.973,A -85,B 0,C 180,E1 -22497.748,E2 -22497.748} C_VEL
LIN {X 0,Y 179.376,Z 294.944,A -85,B 0,C 180,E1 -22499.996,E2 -22499.996} C_VEL
LIN {X 0,Y 178.881,Z 295.017,A -85,B 0,C 180,E1 -22504.503,E2 -22504.503} C_VEL
LIN {X 0,Y 178.966,Z 294.996,A -85,B 0,C 180,E1 -22509.033,E2 -22509.033} C_VEL
LIN {X 0,Y 178.686,Z 295.036,A -85,B 0,C 180,E1 -22513.645,E2 -22513.645} C_VEL
LIN {X 0,Y 178.627,Z 295.043,A -85,B 0,C 180,E1 -22519.211,E2 -22519.211} C_VEL
LIN {X 0,Y 178.536,Z 295.055,A -85,B 0,C 180,E1 -22525.119,E2 -22525.119} C_VEL
LIN {X 0,Y 178.479,Z 295.063,A -85,B 0,C 180,E1 -22530.785,E2 -22530.785} C_VEL
LIN {X 0,Y 178.485,Z 295.063,A -85,B 0,C 180,E1 -22534.215,E2 -22534.215} C_VEL
LIN {X 0,Y 178.493,Z 295.063,A -85,B 0,C 180,E1 -22539.043,E2 -22539.043} C_VEL
LIN {X 0,Y 178.517,Z 295.06,A -85,B 0,C 180,E1 -22542.004,E2 -22542.004} C_VEL
LIN {X 0,Y 178.526,Z 295.058,A -85,B 0,C 180,E1 -22545.114,E2 -22545.114} C_VEL
LIN {X 0,Y 178.513,Z 295.06,A -85,B 0,C 180,E1 -22548.412,E2 -22548.412} C_VEL
LIN {X 0,Y 178.461,Z 295.064,A -85,B 0,C 180,E1 -22553.789,E2 -22553.789} C_VEL
LIN {X 0,Y 178.483,Z 295.065,A -85,B 0,C 180,E1 -22556.543,E2 -22556.543} C_VEL
LIN {X 0,Y 178.514,Z 295.06,A -85,B 0,C 180,E1 -22560.002,E2 -22560.002} C_VEL
LIN {X 0,Y 178.51,Z 295.061,A -85,B 0,C 180,E1 -22564.881,E2 -22564.881} C_VEL
LIN {X 0,Y 178.388,Z 295.076,A -85,B 0,C 180,E1 -22569.23,E2 -22569.23} C_VEL
LIN {X 0,Y 178.386,Z 295.072,A -85,B 0,C 180,E1 -22571.625,E2 -22571.625} C_VEL
LIN {X 0,Y 177.819,Z 295.14,A -85,B 0,C 180,E1 -22577.442,E2 -22577.442} C_VEL
LIN {X 0,Y 177.773,Z 295.315,A -85,B 0,C 180,E1 -22578.271,E2 -22578.271} C_VEL
LIN {X 0,Y 180.515,Z 306.369,A -85,B 0,C 180,E1 -22579.66,E2 -22579.66} C_VEL
LIN {X 0,Y 182.013,Z 315.931,A -85,B 0,C 180,E1 -22581.112,E2 -22581.112} C_VEL
LIN {X 0,Y 182.711,Z 323.847,A -85,B 0,C 180,E1 -22582.538,E2 -22582.538} C_VEL
LIN {X 0,Y 182.81,Z 328.118,A -85,B 0,C 180,E1 -22583.374,E2 -22583.374} C_VEL
LIN {X 0,Y 181.218,Z 337.685,A -85,B 0,C 180,E1 -22585.549,E2 -22585.549} C_VEL
LIN {X 0,Y 179.966,Z 345.339,A -85,B 0,C 180,E1 -22587.759,E2 -22587.759} C_VEL
LIN {X 0,Y 178.818,Z 351.65,A -85,B 0,C 180,E1 -22589.997,E2 -22589.997} C_VEL
LIN {X 0,Y 177.961,Z 356.881,A -85,B 0,C 180,E1 -22592.26,E2 -22592.26} C_VEL
LIN {X 0,Y 177.284,Z 361.245,A -85,B 0,C 180,E1 -22594.544,E2 -22594.544} C_VEL
LIN {X 0,Y 176.707,Z 364.879,A -85,B 0,C 180,E1 -22596.85,E2 -22596.85} C_VEL
LIN {X 0,Y 176.134,Z 369.049,A -85,B 0,C 180,E1 -22600.341,E2 -22600.341} C_VEL
LIN {X 0,Y 176.049,Z 370.218,A -85,B 0,C 180,E1 -22601.511,E2 -22601.511} C_VEL
LIN {X 0,Y 175.987,Z 371.938,A -85,B 0,C 180,E1 -22603.86,E2 -22603.86} C_VEL
LIN {X 0,Y 176.205,Z 373.39,A -85,B 0,C 180,E1 -22606.833,E2 -22606.833} C_VEL
LIN {X 0,Y 177.062,Z 374.002,A -85,B 0,C 180,E1 -22610.927,E2 -22610.927} C_VEL
LIN {X 0,Y 177.888,Z 373.678,A -85,B 0,C 180,E1 -22613.268,E2 -22613.268} C_VEL
LIN {X 0,Y 178.925,Z 372.746,A -85,B 0,C 180,E1 -22615.595,E2 -22615.595} C_VEL
LIN {X 0,Y 180.888,Z 370.389,A -85,B 0,C 180,E1 -22619.052,E2 -22619.052} C_VEL
LIN {X 0,Y 183.417,Z 366.587,A -85,B 0,C 180,E1 -22622.438,E2 -22622.438} C_VEL
LIN {X 0,Y 186.52,Z 361.32,A -85,B 0,C 180,E1 -22625.731,E2 -22625.731} C_VEL
LIN {X 0,Y 189.554,Z 355.599,A -85,B 0,C 180,E1 -22628.387,E2 -22628.387} C_VEL
LIN {X 0,Y 192.945,Z 348.217,A -85,B 0,C 180,E1 -22630.965,E2 -22630.965} C_VEL
LIN {X 0,Y 193.461,Z 346.518,A -85,B 0,C 180,E1 -22631.493,E2 -22631.493} C_VEL
LIN {X 0,Y 193.457,Z 340.397,A -85,B 0,C 180,E1 -22633.645,E2 -22633.645} C_VEL
LIN {X 0,Y 192.902,Z 333.958,A -85,B 0,C 180,E1 -22635.729,E2 -22635.729} C_VEL
LIN {X 0,Y 191.884,Z 327.378,A -85,B 0,C 180,E1 -22637.713,E2 -22637.713} C_VEL
LIN {X 0,Y 190.145,Z 320.683,A -85,B 0,C 180,E1 -22639.704,E2 -22639.704} C_VEL
LIN {X 0,Y 187.264,Z 313.107,A -85,B 0,C 180,E1 -22642.006,E2 -22642.006} C_VEL
LIN {X 0,Y 183.707,Z 305.839,A -85,B 0,C 180,E1 -22644.315,E2 -22644.315} C_VEL
LIN {X 0,Y 181.766,Z 302.304,A -85,B 0,C 180,E1 -22645.427,E2 -22645.427} C_VEL
LIN {X 0,Y 179.281,Z 298.602,A -85,B 0,C 180,E1 -22646.804,E2 -22646.804} C_VEL
LIN {X 0,Y 178.753,Z 296.959,A -85,B 0,C 180,E1 -22647.281,E2 -22647.281} C_VEL
LIN {X 0,Y 178.522,Z 295.356,A -85,B 0,C 180,E1 -22651.814,E2 -22651.814} C_VEL
LIN {X 0,Y 178.505,Z 295.064,A -85,B 0,C 180,E1 -22654.889,E2 -22654.889} C_VEL
LIN {X 0,Y 178.608,Z 295.05,A -85,B 0,C 180,E1 -22660.788,E2 -22660.788} C_VEL
LIN {X 0,Y 178.652,Z 295.045,A -85,B 0,C 180,E1 -22664.02,E2 -22664.02} C_VEL
LIN {X 0,Y 178.821,Z 295.015,A -85,B 0,C 180,E1 -22669.261,E2 -22669.261} C_VEL
LIN {X 0,Y 178.893,Z 295.005,A -85,B 0,C 180,E1 -22673.236,E2 -22673.236} C_VEL
LIN {X 0,Y 179.141,Z 294.974,A -85,B 0,C 180,E1 -22677.756,E2 -22677.756} C_VEL
LIN {X 0,Y 179.36,Z 294.957,A -85,B 0,C 180,E1 -22680.004,E2 -22680.004} C_VEL
LIN {X 0,Y 178.867,Z 295.017,A -85,B 0,C 180,E1 -22684.511,E2 -22684.511} C_VEL
LIN {X 0,Y 178.97,Z 295.004,A -85,B 0,C 180,E1 -22689.041,E2 -22689.041} C_VEL
LIN {X 0,Y 178.681,Z 295.041,A -85,B 0,C 180,E1 -22693.654,E2 -22693.654} C_VEL
LIN {X 0,Y 178.644,Z 295.044,A -85,B 0,C 180,E1 -22698.348,E2 -22698.348} C_VEL
LIN {X 0,Y 178.492,Z 295.067,A -85,B 0,C 180,E1 -22703.192,E2 -22703.192} C_VEL
LIN {X 0,Y 178.577,Z 295.79,A -85,B 0,C 180,E1 -22705.656,E2 -22705.656} C_VEL
LIN {X 0,Y 178.982,Z 297.87,A -85,B 0,C 180,E1 -22710.699,E2 -22710.699} C_VEL
LIN {X 0,Y 179.449,Z 300.416,A -85,B 0,C 180,E1 -22715.981,E2 -22715.981} C_VEL
LIN {X 0,Y 179.687,Z 301.922,A -85,B 0,C 180,E1 -22718.745,E2 -22718.745} C_VEL
LIN {X 0,Y 179.966,Z 303.886,A -85,B 0,C 180,E1 -22722.104,E2 -22722.104} C_VEL
LIN {X 0,Y 180.523,Z 307.286,A -85,B 0,C 180,E1 -22727.462,E2 -22727.462} C_VEL
LIN {X 0,Y 181.644,Z 310.395,A -85,B 0,C 180,E1 -22728.194,E2 -22728.194} C_VEL
LIN {X 0,Y 183.486,Z 313.248,A -85,B 0,C 180,E1 -22729.156,E2 -22729.156} C_VEL
LIN {X 0,Y 185.476,Z 317.368,A -85,B 0,C 180,E1 -22730.278,E2 -22730.278} C_VEL
LIN {X 0,Y 187.753,Z 323.146,A -85,B 0,C 180,E1 -22731.825,E2 -22731.825} C_VEL
LIN {X 0,Y 189.159,Z 328.176,A -85,B 0,C 180,E1 -22733.023,E2 -22733.023} C_VEL
LIN {X 0,Y 190.452,Z 337.712,A -85,B 0,C 180,E1 -22735.236,E2 -22735.236} C_VEL
LIN {X 0,Y 190.873,Z 345.904,A -85,B 0,C 180,E1 -22737.283,E2 -22737.283} C_VEL
LIN {X 0,Y 190.691,Z 354.061,A -85,B 0,C 180,E1 -22739.555,E2 -22739.555} C_VEL
LIN {X 0,Y 190.176,Z 359.686,A -85,B 0,C 180,E1 -22741.291,E2 -22741.291} C_VEL
LIN {X 0,Y 189.058,Z 366.071,A -85,B 0,C 180,E1 -22743.511,E2 -22743.511} C_VEL
LIN {X 0,Y 187.73,Z 370.266,A -85,B 0,C 180,E1 -22745.095,E2 -22745.095} C_VEL
LIN {X 0,Y 184.713,Z 376.013,A -85,B 0,C 180,E1 -22747.64,E2 -22747.64} C_VEL
LIN {X 0,Y 182.615,Z 379.806,A -85,B 0,C 180,E1 -22749.738,E2 -22749.738} C_VEL
LIN {X 0,Y 180.037,Z 384.166,A -85,B 0,C 180,E1 -22752.979,E2 -22752.979} C_VEL
LIN {X 0,Y 178.159,Z 387.262,A -85,B 0,C 180,E1 -22756.312,E2 -22756.312} C_VEL
LIN {X 0,Y 177.26,Z 388.707,A -85,B 0,C 180,E1 -22758.569,E2 -22758.569} C_VEL
LIN {X 0,Y 176.634,Z 389.677,A -85,B 0,C 180,E1 -22760.845,E2 -22760.845} C_VEL
LIN {X 0,Y 176.249,Z 390.065,A -85,B 0,C 180,E1 -22763.133,E2 -22763.133} C_VEL
LIN {X 0,Y 176.114,Z 389.889,A -85,B 0,C 180,E1 -22766.114,E2 -22766.114} C_VEL
LIN {X 0,Y 176.418,Z 388.415,A -85,B 0,C 180,E1 -22770.003,E2 -22770.003} C_VEL
LIN {X 0,Y 176.207,Z 386.03,A -85,B 0,C 180,E1 -22773.13,E2 -22773.13} C_VEL
LIN {X 0,Y 176.28,Z 383.288,A -85,B 0,C 180,E1 -22775.723,E2 -22775.723} C_VEL
LIN {X 0,Y 176.604,Z 378.858,A -85,B 0,C 180,E1 -22778.824,E2 -22778.824} C_VEL
LIN {X 0,Y 177.129,Z 374.102,A -85,B 0,C 180,E1 -22781.446,E2 -22781.446} C_VEL
LIN {X 0,Y 177.891,Z 369.051,A -85,B 0,C 180,E1 -22783.715,E2 -22783.715} C_VEL
LIN {X 0,Y 178.839,Z 362.947,A -85,B 0,C 180,E1 -22785.97,E2 -22785.97} C_VEL
LIN {X 0,Y 179.24,Z 360.677,A -85,B 0,C 180,E1 -22786.707,E2 -22786.707} C_VEL
LIN {X 0,Y 179.376,Z 357.891,A -85,B 0,C 180,E1 -22787.592,E2 -22787.592} C_VEL
LIN {X 0,Y 178.901,Z 355.066,A -85,B 0,C 180,E1 -22788.458,E2 -22788.458} C_VEL
LIN {X 0,Y 176.875,Z 349.329,A -85,B 0,C 180,E1 -22790.112,E2 -22790.112} C_VEL
LIN {X 0,Y 174.059,Z 341.63,A -85,B 0,C 180,E1 -22792.03,E2 -22792.03} C_VEL
LIN {X 0,Y 173.275,Z 336.539,A -85,B 0,C 180,E1 -22793.052,E2 -22793.052} C_VEL
LIN {X 0,Y 172.786,Z 325.785,A -85,B 0,C 180,E1 -22794.789,E2 -22794.789} C_VEL
LIN {X 0,Y 171.641,Z 315.451,A -85,B 0,C 180,E1 -22796.105,E2 -22796.105} C_VEL
LIN {X 0,Y 170.724,Z 309.008,A -85,B 0,C 180,E1 -22796.786,E2 -22796.786} C_VEL
LIN {X 0,Y 172.048,Z 304.417,A -85,B 0,C 180,E1 -22802.079,E2 -22802.079} C_VEL
LIN {X 0,Y 172.565,Z 302.125,A -85,B 0,C 180,E1 -22804.766,E2 -22804.766} C_VEL
LIN {X 0,Y 172.147,Z 298.693,A -85,B 0,C 180,E1 -22809.128,E2 -22809.128} C_VEL
LIN {X 0,Y 171.558,Z 295.927,A -85,B 0,C 180,E1 -22813.006,E2 -22813.006} C_VEL
LIN {X 0,Y 171.352,Z 295.952,A -85,B 0,C 180,E1 -22818.982,E2 -22818.982} C_VEL
LIN {X 0,Y 171.399,Z 295.942,A -85,B 0,C 180,E1 -22822.04,E2 -22822.04} C_VEL
LIN {X 0,Y 171.411,Z 295.945,A -85,B 0,C 180,E1 -22825.091,E2 -22825.091} C_VEL
LIN {X 0,Y 171.462,Z 295.934,A -85,B 0,C 180,E1 -22830.533,E2 -22830.533} C_VEL
LIN {X 0,Y 171.454,Z 295.935,A -85,B 0,C 180,E1 -22835.797,E2 -22835.797} C_VEL
LIN {X 0,Y 171.522,Z 295.929,A -85,B 0,C 180,E1 -22840.861,E2 -22840.861} C_VEL
LIN {X 0,Y 171.568,Z 295.921,A -85,B 0,C 180,E1 -22845.768,E2 -22845.768} C_VEL
LIN {X 0,Y 171.854,Z 295.886,A -85,B 0,C 180,E1 -22850.581,E2 -22850.581} C_VEL
LIN {X 0,Y 171.82,Z 295.892,A -85,B 0,C 180,E1 -22855.303,E2 -22855.303} C_VEL
LIN {X 0,Y 172.339,Z 295.82,A -85,B 0,C 180,E1 -22859.996,E2 -22859.996} C_VEL
LIN {X 0,Y 171.83,Z 295.894,A -85,B 0,C 180,E1 -22864.688,E2 -22864.688} C_VEL
LIN {X 0,Y 171.895,Z 295.876,A -85,B 0,C 180,E1 -22869.408,E2 -22869.408} C_VEL
LIN {X 0,Y 171.599,Z 295.921,A -85,B 0,C 180,E1 -22874.221,E2 -22874.221} C_VEL
LIN {X 0,Y 171.548,Z 295.925,A -85,B 0,C 180,E1 -22879.557,E2 -22879.557} C_VEL
LIN {X 0,Y 171.471,Z 295.937,A -85,B 0,C 180,E1 -22885.611,E2 -22885.611} C_VEL
LIN {X 0,Y 171.442,Z 295.939,A -85,B 0,C 180,E1 -22890.581,E2 -22890.581} C_VEL
LIN {X 0,Y 171.439,Z 295.94,A -85,B 0,C 180,E1 -22895.018,E2 -22895.018} C_VEL
LIN {X 0,Y 171.444,Z 295.941,A -85,B 0,C 180,E1 -22898.839,E2 -22898.839} C_VEL
LIN {X 0,Y 171.451,Z 295.939,A -85,B 0,C 180,E1 -22904.168,E2 -22904.168} C_VEL
LIN {X 0,Y 171.429,Z 295.943,A -85,B 0,C 180,E1 -22909.005,E2 -22909.005} C_VEL
LIN {X 0,Y 171.436,Z 295.941,A -85,B 0,C 180,E1 -22912.05,E2 -22912.05} C_VEL
LIN {X 0,Y 171.411,Z 295.943,A -85,B 0,C 180,E1 -22917.788,E2 -22917.788} C_VEL
LIN {X 0,Y 171.44,Z 295.943,A -85,B 0,C 180,E1 -22920.529,E2 -22920.529} C_VEL
LIN {X 0,Y 171.425,Z 295.943,A -85,B 0,C 180,E1 -22925.794,E2 -22925.794} C_VEL
LIN {X 0,Y 171.354,Z 295.95,A -85,B 0,C 180,E1 -22930.842,E2 -22930.842} C_VEL
LIN {X 0,Y 170.89,Z 296.008,A -85,B 0,C 180,E1 -22935.711,E2 -22935.711} C_VEL
LIN {X 0,Y 170.819,Z 296.199,A -85,B 0,C 180,E1 -22937.459,E2 -22937.459} C_VEL
LIN {X 0,Y 173.445,Z 306.283,A -85,B 0,C 180,E1 -22938.808,E2 -22938.808} C_VEL
LIN {X 0,Y 174.87,Z 314.939,A -85,B 0,C 180,E1 -22940.161,E2 -22940.161} C_VEL
LIN {X 0,Y 175.752,Z 323.053,A -85,B 0,C 180,E1 -22941.662,E2 -22941.662} C_VEL
LIN {X 0,Y 175.937,Z 328.703,A -85,B 0,C 180,E1 -22942.826,E2 -22942.826} C_VEL
LIN {X 0,Y 174.288,Z 338.205,A -85,B 0,C 180,E1 -22945.081,E2 -22945.081} C_VEL
LIN {X 0,Y 173.147,Z 344.968,A -85,B 0,C 180,E1 -22947.089,E2 -22947.089} C_VEL
LIN {X 0,Y 171.933,Z 351.395,A -85,B 0,C 180,E1 -22949.411,E2 -22949.411} C_VEL
LIN {X 0,Y 170.997,Z 356.728,A -85,B 0,C 180,E1 -22951.763,E2 -22951.763} C_VEL
LIN {X 0,Y 170.14,Z 362.15,A -85,B 0,C 180,E1 -22954.736,E2 -22954.736} C_VEL
LIN {X 0,Y 169.552,Z 365.67,A -85,B 0,C 180,E1 -22957.14,E2 -22957.14} C_VEL
LIN {X 0,Y 169.02,Z 369.732,A -85,B 0,C 180,E1 -22960.781,E2 -22960.781} C_VEL
LIN {X 0,Y 168.935,Z 372.517,A -85,B 0,C 180,E1 -22964.451,E2 -22964.451} C_VEL
LIN {X 0,Y 169.155,Z 373.712,A -85,B 0,C 180,E1 -22967.156,E2 -22967.156} C_VEL
LIN {X 0,Y 169.521,Z 374.198,A -85,B 0,C 180,E1 -22969.366,E2 -22969.366} C_VEL
LIN {X 0,Y 170.207,Z 374.292,A -85,B 0,C 180,E1 -22971.812,E2 -22971.812} C_VEL
LIN {X 0,Y 171.135,Z 373.891,A -85,B 0,C 180,E1 -22974.243,E2 -22974.243} C_VEL
LIN {X 0,Y 172.296,Z 372.93,A -85,B 0,C 180,E1 -22976.656,E2 -22976.656} C_VEL
LIN {X 0,Y 174.464,Z 370.383,A -85,B 0,C 180,E1 -22980.231,E2 -22980.231} C_VEL
LIN {X 0,Y 177.103,Z 366.669,A -85,B 0,C 180,E1 -22983.565,E2 -22983.565} C_VEL
LIN {X 0,Y 179.384,Z 363.037,A -85,B 0,C 180,E1 -22985.988,E2 -22985.988} C_VEL
LIN {X 0,Y 181.784,Z 358.839,A -85,B 0,C 180,E1 -22988.208,E2 -22988.208} C_VEL
LIN {X 0,Y 184.636,Z 353.513,A -85,B 0,C 180,E1 -22990.43,E2 -22990.43} C_VEL
LIN {X 0,Y 186.631,Z 349.448,A -85,B 0,C 180,E1 -22991.868,E2 -22991.868} C_VEL
LIN {X 0,Y 187.122,Z 346.195,A -85,B 0,C 180,E1 -22993.044,E2 -22993.044} C_VEL
LIN {X 0,Y 187.044,Z 339.31,A -85,B 0,C 180,E1 -22995.549,E2 -22995.549} C_VEL
LIN {X 0,Y 186.288,Z 332.088,A -85,B 0,C 180,E1 -22997.967,E2 -22997.967} C_VEL
LIN {X 0,Y 184.859,Z 325.275,A -85,B 0,C 180,E1 -23000.166,E2 -23000.166} C_VEL
LIN {X 0,Y 182.356,Z 317.801,A -85,B 0,C 180,E1 -23002.633,E2 -23002.633} C_VEL
LIN {X 0,Y 179.525,Z 311.536,A -85,B 0,C 180,E1 -23004.805,E2 -23004.805} C_VEL
LIN {X 0,Y 177.43,Z 307.233,A -85,B 0,C 180,E1 -23006.327,E2 -23006.327} C_VEL
LIN {X 0,Y 175.153,Z 303.658,A -85,B 0,C 180,E1 -23007.718,E2 -23007.718} C_VEL
LIN {X 0,Y 174.356,Z 302.229,A -85,B 0,C 180,E1 -23008.235,E2 -23008.235} C_VEL
LIN {X 0,Y 172.319,Z 299.364,A -85,B 0,C 180,E1 -23009.49,E2 -23009.49} C_VEL
LIN {X 0,Y 171.701,Z 297.449,A -85,B 0,C 180,E1 -23010.069,E2 -23010.069} C_VEL
LIN {X 0,Y 171.487,Z 296.129,A -85,B 0,C 180,E1 -23014.363,E2 -23014.363} C_VEL
LIN {X 0,Y 171.564,Z 295.927,A -85,B 0,C 180,E1 -23020.875,E2 -23020.875} C_VEL
LIN {X 0,Y 171.584,Z 295.917,A -85,B 0,C 180,E1 -23025.778,E2 -23025.778} C_VEL
LIN {X 0,Y 171.833,Z 295.887,A -85,B 0,C 180,E1 -23030.588,E2 -23030.588} C_VEL
LIN {X 0,Y 171.8,Z 295.896,A -85,B 0,C 180,E1 -23035.311,E2 -23035.311} C_VEL
LIN {X 0,Y 172.323,Z 295.833,A -85,B 0,C 180,E1 -23040.004,E2 -23040.004} C_VEL
LIN {X 0,Y 171.816,Z 295.893,A -85,B 0,C 180,E1 -23044.697,E2 -23044.697} C_VEL
LIN {X 0,Y 171.903,Z 295.884,A -85,B 0,C 180,E1 -23049.416,E2 -23049.416} C_VEL
LIN {X 0,Y 171.603,Z 295.923,A -85,B 0,C 180,E1 -23054.229,E2 -23054.229} C_VEL
LIN {X 0,Y 171.536,Z 295.932,A -85,B 0,C 180,E1 -23059.564,E2 -23059.564} C_VEL
LIN {X 0,Y 171.462,Z 296.116,A -85,B 0,C 180,E1 -23061.652,E2 -23061.652} C_VEL
LIN {X 0,Y 171.727,Z 297.896,A -85,B 0,C 180,E1 -23066.759,E2 -23066.759} C_VEL
LIN {X 0,Y 172.143,Z 300.083,A -85,B 0,C 180,E1 -23072.06,E2 -23072.06} C_VEL
LIN {X 0,Y 172.485,Z 301.653,A -85,B 0,C 180,E1 -23075.427,E2 -23075.427} C_VEL
LIN {X 0,Y 172.846,Z 304.429,A -85,B 0,C 180,E1 -23080.589,E2 -23080.589} C_VEL
LIN {X 0,Y 173.287,Z 306.895,A -85,B 0,C 180,E1 -23084.706,E2 -23084.706} C_VEL
LIN {X 0,Y 174.32,Z 309.83,A -85,B 0,C 180,E1 -23085.449,E2 -23085.449} C_VEL
LIN {X 0,Y 176.409,Z 313.121,A -85,B 0,C 180,E1 -23086.683,E2 -23086.683} C_VEL
LIN {X 0,Y 178.457,Z 317.153,A -85,B 0,C 180,E1 -23087.944,E2 -23087.944} C_VEL
LIN {X 0,Y 182.126,Z 325.531,A -85,B 0,C 180,E1 -23090.518,E2 -23090.518} C_VEL
LIN {X 0,Y 183.676,Z 332.036,A -85,B 0,C 180,E1 -23092.255,E2 -23092.255} C_VEL
LIN {X 0,Y 184.529,Z 340.494,A -85,B 0,C 180,E1 -23094.393,E2 -23094.393} C_VEL
LIN {X 0,Y 184.673,Z 349.53,A -85,B 0,C 180,E1 -23096.855,E2 -23096.855} C_VEL
LIN {X 0,Y 184.044,Z 358.395,A -85,B 0,C 180,E1 -23099.608,E2 -23099.608} C_VEL
LIN {X 0,Y 182.895,Z 365.339,A -85,B 0,C 180,E1 -23102.111,E2 -23102.111} C_VEL
LIN {X 0,Y 181.307,Z 370.431,A -85,B 0,C 180,E1 -23104.149,E2 -23104.149} C_VEL
